# B&R Automation Studio project TD52 (part 136)

#### MSC_MB.st
```iecst
(********************************************************************
 * COPYRIGHT -- INNIO, MSC
 ********************************************************************
 * Library: MSC_MB
 * File: MSC_MB.st
 * Author: Hohensinner Michael
 * Created: April 29, 2021
 ********************************************************************
 * Functions and function blocks of library MSC_MB
 ********************************************************************)
(* ModBus Master function block 4 easy use *)
FUNCTION MSC_MB_RegUpdate
	MSC_MB_RegUpdate := 0;
	bError := FALSE;
	IF tSlave.bSkip THEN
		iWrite	:=	0;
		iRead	:=	0;
		FOR x:=0 TO _MB_CMD_MAX DO
			tSlave.tLine[x].tIF.bExec	:=	FALSE;
		END_FOR
		RETURN;
	END_IF
	FOR x:=0 TO _MB_CMD_MAX DO
		IF tSlave.tLine[x].tDef.pDest > 0 THEN
			CASE tSlave.tLine[x].tDef.iFC OF
				1,2,5,15:	iByteSize := 2 * REAL_TO_UINT(brmceil((UINT_TO_REAL(tSlave.tLine[x].tDef.iLen) + USINT_TO_REAL(tSlave.tLine[x].tDef.iBitOffs))/16.0));		//Bitwise
				3,4,6,16:	iByteSize := 2 * REAL_TO_UINT(brmceil(UINT_TO_REAL(tSlave.tLine[x].tDef.iLen) + USINT_TO_REAL(tSlave.tLine[x].tDef.iBitOffs)/16.0));		//Wordwise
				ELSE
					MSC_MB_RegUpdate := 1;
					RETURN;	// Wrong function code
			END_CASE
			IF SIZEOF(iTemp) < iByteSize THEN
				MSC_MB_RegUpdate := 2;
				RETURN;	// To small temporary register
			END_IF
			IF iByteSize < 2 THEN
				MSC_MB_RegUpdate := 3;
				RETURN;	// To small, at least a word to copy (should not happen)
			END_IF
			brsmemcpy(ADR(iTemp),tSlave.tLine[x].tDef.pDest,iByteSize);

			CASE tSlave.tLine[x].tDef.iFC OF
				1..4:
					IF GET_BIT_UINT_ARRAY(x,ADR(iRead)) THEN
						tSlave.tLine[x].tIF.bExec	:=	bEnaRead;
					END_IF
				5,6,15,16:
					IF GET_BIT_UINT_ARRAY(x,ADR(iWrite)) THEN
						tSlave.tLine[x].tIF.bExec	:=	bEnaWrite;
					END_IF
			END_CASE
			IF tSlave.tLine[x].tIF.iStatus <> 0 AND tSlave.tLine[x].tIF.iStatus <> 65535 THEN
				bError := TRUE;
				iError := tSlave.tLine[x].tIF.iStatus;
			END_IF

			CASE tSlave.tLine[x].tDef.iFC OF
				1,2:
					FOR i:= 0 TO  MAX(0,tSlave.tLine[x].tDef.iLen-1) DO
						IF i > _MB_BIN_MAX THEN
							MSC_MB_RegUpdate := tSlave.tLine[x].tDef.iFC * 10 + 1;
							RETURN;	// OUT OF BINARY BOUNDS
						END_IF
						SET_BIT_UINT_ARRAY(tSlave.tLine[x].tIF.bData[i],i + tSlave.tLine[x].tDef.iBitOffs,ADR(iTemp));
					END_FOR
					brsmemcpy(tSlave.tLine[x].tDef.pDest,ADR(iTemp),iByteSize);
				3,4:
					IF tSlave.tLine[x].tDef.iBitOffs = 0 THEN
						brsmemcpy(tSlave.tLine[x].tDef.pDest,ADR(tSlave.tLine[x].tIF.iData),tSlave.tLine[x].tDef.iLen*2);
					ELSE
						FOR i:= 0 TO MAX(0,tSlave.tLine[x].tDef.iLen*16-1) DO
							IF i/16 > _MB_REG_MAX THEN
								MSC_MB_RegUpdate := tSlave.tLine[x].tDef.iFC * 10 + 1;
								RETURN;	// OUT OF REGISTER BOUNDS
							END_IF
							SET_BIT_UINT_ARRAY(GET_BIT_UINT_ARRAY(i,ADR(tSlave.tLine[x].tIF.iData)),i + tSlave.tLine[x].tDef.iBitOffs,ADR(iTemp));
						END_FOR
						brsmemcpy(tSlave.tLine[x].tDef.pDest,ADR(iTemp),iByteSize);
					END_IF

				5,15:
					IF tSlave.tLine[x].tDef.iFC = 5 THEN
						tSlave.tLine[x].tIF.bData[0] := GET_BIT_UINT_ARRAY(tSlave.tLine[x].tDef.iBitOffs,ADR(iTemp));
					ELSIF tSlave.tLine[x].tDef.iFC = 15 THEN
						FOR i:= 0 TO MAX(0, tSlave.tLine[x].tDef.iLen-1) DO
							IF i > _MB_BIN_MAX THEN
								MSC_MB_RegUpdate := tSlave.tLine[x].tDef.iFC * 10 + 1;
								RETURN;	// OUT OF BINARY BOUNDS
							END_IF
							tSlave.tLine[x].tIF.bData[i]	:=	GET_BIT_UINT_ARRAY(i+tSlave.tLine[x].tDef.iBitOffs,ADR(iTemp));
						END_FOR
					END_IF

				6,16:
					IF tSlave.tLine[x].tDef.iBitOffs = 0 THEN
						FOR i:= 0 TO MAX(0,tSlave.tLine[x].tDef.iLen-1) DO
							IF i > _MB_REG_MAX THEN
								MSC_MB_RegUpdate := tSlave.tLine[x].tDef.iFC * 10;
								RETURN;	// OUT OF REGISTER BOUNDS
							END_IF
							tSlave.tLine[x].tIF.iData[i]	:=	iTemp[i];
						END_FOR
					ELSE
						FOR i:= 0 TO MAX(0,tSlave.tLine[x].tDef.iLen*16-1) DO
							IF i/16 > _MB_REG_MAX THEN
								MSC_MB_RegUpdate := tSlave.tLine[x].tDef.iFC * 10 + 1;
								RETURN;	// OUT OF REGISTER BOUNDS
							END_IF
							SET_BIT_UINT_ARRAY(GET_BIT_UINT_ARRAY(i+tSlave.tLine[x].tDef.iBitOffs,ADR(iTemp)),i,ADR(tSlave.tLine[x].tIF.iData));
						END_FOR
					END_IF
			END_CASE
		END_IF
	END_FOR
	IF NOT bError THEN
		iError	:=	0;
	END_IF
	iWrite	:=	0;
	iRead	:=	0;
	RETURN;
END_FUNCTION

FUNCTION_BLOCK MSC_MBMaster
	IF bEnable THEN
		CASE eState OF
			_MB_DEFAULT:
				IF tCmd.bOpen THEN
					tCmd.bOpen	:=	FALSE;
					eState		:=	_MB_OPEN;
				END_IF
			_MB_OPEN:
				xMBMOpen.enable		:= TRUE;
				xMBMOpen.pDevice	:= ADR(tCfg.sDevice);
				xMBMOpen.pMode		:= ADR(tCfg.sMode);
				xMBMOpen.pConfig	:= ADR(tCfg.sFile);
				xMBMOpen.timeout	:= tCfg.iTimeOut;
				xMBMOpen.ascii		:= BOOL_TO_USINT(tCfg.bASCII);
				xMBMOpen();
				IF (xMBMOpen.status <> ERR_FUB_BUSY) THEN
					IF (xMBMOpen.status = ERR_OK) THEN
						xMBMaster.enable	:=	TRUE;
						xMBMaster.ident		:=	xMBMOpen.ident;
						eState				:=	_MB_RUN;
					ELSE
						eError				:=	eState;
						iError				:=	xMBMOpen.status;
						eState				:=	_MB_ERROR;
					END_IF
				END_IF
			_MB_RUN:
				IF tCmd.bClose THEN
					tCmd.bClose			:=	FALSE;
					xMBMaster.enable	:=	FALSE;
					xMBMClose.enable	:=	TRUE;
					xMBMClose.ident		:=	xMBMOpen.ident;
					eState 				:=	_MB_CLOSE;
				ELSE
					xMBMaster();
				END_IF
			_MB_CLOSE:
				xMBMClose();
				IF (xMBMClose.status <> ERR_FUB_BUSY) THEN
					IF (xMBMClose.status = ERR_OK) THEN
						eState		:=	_MB_DEFAULT;
					ELSE
						eError		:=	eState;
						iError		:=	xMBMOpen.status;
						eState		:=	_MB_ERROR;
					END_IF
				END_IF
			_MB_ERROR:
				IF tCmd.bAckn THEN
					tCmd.bAckn		:=	FALSE;
					eState			:=	_MB_DEFAULT;
				END_IF
		END_CASE
	END_IF
	bExec	:=	xMBMaster.execute;
	iRecNum	:=	xMBMaster.recordnum;
	iStatus	:=	xMBMaster.status;
END_FUNCTION_BLOCK
(* ModBus Slave function block 4 easy use *)
FUNCTION_BLOCK MSC_MBSlave
	IF bEnable THEN
		CASE eState OF
			_MB_DEFAULT:
				IF tCmd.bOpen THEN
					tCmd.bOpen	:=	FALSE;
					eState		:=	_MB_OPEN;
				END_IF
			_MB_OPEN:
				xMBSOpen.enable		:= TRUE;
				xMBSOpen.pDevice	:= ADR(tCfg.sDevice);
				xMBSOpen.pMode		:= ADR(tCfg.sMode);
				xMBSOpen.own_ID		:= tCfg.iID;
				xMBSOpen.timeout	:= tCfg.iTimeOut;
				xMBSOpen.pCoilStat	:= tCfg.pCoilStat;
				xMBSOpen.pHoldingReg:= tCfg.pHoldReg;
				xMBSOpen.pInputReg	:= tCfg.pInReg;
				xMBSOpen.pInputStat	:= tCfg.pInStat;
				xMBSOpen();
				IF (xMBSOpen.status <> ERR_FUB_BUSY) THEN
					IF (xMBSOpen.status = ERR_OK) THEN
						xMBSlave.enable	:=	TRUE;
						xMBSlave.ident		:=	xMBSOpen.ident;
						eState				:=	_MB_RUN;
					ELSE
						eError				:=	eState;
						iError				:=	xMBSOpen.status;
						eState				:=	_MB_ERROR;
					END_IF
				END_IF
			_MB_RUN:
				IF tCmd.bClose THEN
					tCmd.bClose			:=	FALSE;
					xMBSlave.enable		:=	FALSE;
					xMBSClose.enable	:=	TRUE;
					xMBSClose.ident		:=	xMBSOpen.ident;
					eState 				:=	_MB_CLOSE;
				ELSE
					xMBSlave();
				END_IF
			_MB_CLOSE:
				xMBSClose();
				IF (xMBSClose.status <> ERR_FUB_BUSY) THEN
					IF (xMBSClose.status = ERR_OK) THEN
						eState		:=	_MB_DEFAULT;
					ELSE
						eError		:=	eState;
						iError		:=	xMBSOpen.status;
						eState		:=	_MB_ERROR;
					END_IF
				END_IF
			_MB_ERROR:
				IF tCmd.bAckn THEN
					tCmd.bAckn		:=	FALSE;
					eState			:=	_MB_DEFAULT;
				END_IF
		END_CASE
	END_IF
END_FUNCTION_BLOCK

(* ModBus Data Object single line *)
FUNCTION_BLOCK MSC_MB_DataLine
	(* clear old data if previously used *)
	FOR iBegin:=0 TO _MB_DATALINE_MAX DO
		iData[iBegin]	:=	0;
	END_FOR
	bError	:=	FALSE;
	iBegin	:=	0;
	iStrLen	:=	0;
	sData	:=	'';
	(* Execution variable BEGIN *)
	brsstrcat(ADR(sData),ADR('"'));
	IF pName_Module > 0 THEN
		brsstrcat(ADR(sData),pName_Module);
		brsstrcat(ADR(sData),ADR('::'));
	END_IF
	IF pName_Task > 0 THEN
		brsstrcat(ADR(sData),pName_Task);
		brsstrcat(ADR(sData),ADR(':'));
	END_IF
	IF pName_Struct > 0 THEN
		brsstrcat(ADR(sData),pName_Struct);
	ELSE
		brsstrcat(ADR(sData),ADR('tSlave'));
	END_IF
	brsitoa(iIdx_Slave,ADR(sTemp));
	brsstrcat(ADR(sData),ADR('['));
	brsstrcat(ADR(sData),ADR(sTemp));
	brsstrcat(ADR(sData),ADR(']'));

	brsstrcat(ADR(sData),ADR('.tLine'));
	brsitoa(iIdx_Line,ADR(sTemp));
	brsstrcat(ADR(sData),ADR('['));
	brsstrcat(ADR(sData),ADR(sTemp));
	brsstrcat(ADR(sData),ADR('].tIF.bExec"'));

	iStrLen := brsstrlen(ADR(sData))-2;
	IF iStrLen < _MB_DATALINE_MAX THEN
		brsmemcpy(ADR(iData[0]),ADR(sData)+1,iStrLen);
	ELSE
		bError	:=	TRUE;
	END_IF
	(* Execution variable END *)

	(* Spacing *)
	iData[iStrLen] := 0;
	(* Functional code *)
	iData[iStrLen+1] := iFC;
	(* Address of slave *)
	iData[iStrLen+2] := iAdr_Slave;
	iBegin := iStrLen+3;

	(* Data variable BEGIN *)
	sData := '';
	brsstrcat(ADR(sData),ADR('"'));
	IF pName_Module > 0 THEN
		brsstrcat(ADR(sData),pName_Module);
		brsstrcat(ADR(sData),ADR('::'));
	END_IF
	IF pName_Task > 0 THEN
		brsstrcat(ADR(sData),pName_Task);
		brsstrcat(ADR(sData),ADR(':'));
	END_IF
	IF pName_Struct > 0 THEN
		brsstrcat(ADR(sData),pName_Struct);
	ELSE
		brsstrcat(ADR(sData),ADR('tSlave'));
	END_IF

	brsitoa(iIdx_Slave,ADR(sTemp));
	brsstrcat(ADR(sData),ADR('['));
	brsstrcat(ADR(sData),ADR(sTemp));
	brsstrcat(ADR(sData),ADR(']'));

	brsstrcat(ADR(sData),ADR('.tLine'));
	brsitoa(iIdx_Line,ADR(sTemp));
	brsstrcat(ADR(sData),ADR('['));
	brsstrcat(ADR(sData),ADR(sTemp));
	brsstrcat(ADR(sData),ADR('].tIF.'));

	CASE iFC OF
		1,2,15:	brsstrcat(ADR(sData),ADR('bData'));
		3,4,16:	brsstrcat(ADR(sData),ADR('iData'));
		5:	brsstrcat(ADR(sData),ADR('bData[0]'));
		6:	brsstrcat(ADR(sData),ADR('iData[0]'));
		ELSE
			brsstrcat(ADR(sData),ADR('bNA'));	//through error here
	END_CASE
	brsstrcat(ADR(sData),ADR('"'));
	iStrLen := brsstrlen(ADR(sData))-2;
	IF iBegin + iStrLen + 4 < _MB_DATALINE_MAX THEN
		brsmemcpy(ADR(iData[iBegin]),ADR(sData)+1,iStrLen);
		(* Data variable END *)

		(* Spacing *)
		iData[iBegin + iStrLen] := 0;

		(* Offset *)
		iData[iBegin + iStrLen + 1] := UDINT_TO_USINT(iOffset MOD 256);
		iData[iBegin + iStrLen + 2] := UDINT_TO_USINT(iOffset / 256);
		iStrLen	:=	iBegin + iStrLen + 2 + 1;

		(* Length *)
		iData[iStrLen] := UDINT_TO_USINT(iLength MOD 256);
		iData[iStrLen+1] := UDINT_TO_USINT(iLength / 256);
		iStrLen	:=	iStrLen + 2;
	ELSE
		bError	:=	TRUE;
	END_IF

END_FUNCTION_BLOCK

(* ModBus Data Object multiple lines *)
FUNCTION_BLOCK MSC_MB_DataSet
	(* clear old data if previously used *)
	iStrLen	:=	0;
	bError	:=	FALSE;
	FOR i:=0 TO _MB_DATASET_MAX DO
		iData[i]	:=	0;
	END_FOR

	(* handle over static slave data *)
	xLine.pName_Module	:=	pName_Module;
	xLine.pName_Task	:=	pName_Task;
	xLine.pName_Struct	:=	pName_Struct;
	xLine.iIdx_Slave	:=	iIdx_Slave;
	xLine.iAdr_Slave	:=	iAdr_Slave;
	bEmpty	:=	TRUE;

	(* handle over dynamic slave data, execute only if function code is legit *)
	FOR i:= 0 TO _MB_CMD_MAX DO
		IF (tLine[i].tDef.iFC >= 1 AND tLine[i].tDef.iFC <= 6) OR tLine[i].tDef.iFC = 15 OR tLine[i].tDef.iFC = 16	THEN
			xLine.iIdx_Line	:=	UDINT_TO_USINT(i);
			xLine.iFC		:=	tLine[i].tDef.iFC;
			xLine.iOffset	:=	tLine[i].tDef.iOffs;
			xLine.iLength	:=	tLine[i].tDef.iLen;

			xLine();

			IF iStrLen + xLine.iStrLen < _MB_DATASET_MAX AND NOT xLine.bError THEN
				brsmemcpy(ADR(iData)+iStrLen,ADR(xLine.iData),xLine.iStrLen);
				iStrLen	:=	iStrLen + xLine.iStrLen;
				bEmpty	:=	FALSE;
			ELSE
				bError	:=	TRUE;
			END_IF
		END_IF
	END_FOR

END_FUNCTION_BLOCK

(* ModBus Data Object creator *)
FUNCTION_BLOCK MSC_MB_DOCreate

	CASE eState OF
		_MB_DEFAULT:
			xDatObjInfo.enable		:=	TRUE;
			xDatObjInfo.pName 		:=	pName;
			xDatObjDelete.enable	:=	TRUE;
			xDatObjCreate.enable	:=	TRUE;
			xDatObjCreate.pName		:=	pName;
			xDatObjCreate.pCpyData	:=	pCpyData;
			xDatObjCreate.MemType	:=	iMemType;
			xDatObjCreate.len		:=	iLen;
			IF bEnable THEN
				eState	:=	_MB_INFO;
			END_IF
			bDone := FALSE;
		_MB_INFO:
			xDatObjInfo();
			IF	xDatObjInfo.status = ERR_OK THEN				eState	:=	_MB_DELETE;
			ELSIF xDatObjInfo.status = doERR_MODULNOTFOUND THEN	eState	:=	_MB_CREATE;
			ELSIF xDatObjInfo.status <>  ERR_FUB_BUSY THEN		eState	:=	_MB_ERROR;
			END_IF
		_MB_DELETE:
			xDatObjDelete.ident		:=	xDatObjInfo.ident;
			xDatObjDelete();
			IF	xDatObjDelete.status = ERR_OK THEN				eState	:=	_MB_CREATE;
			ELSIF	xDatObjDelete.status <>  ERR_FUB_BUSY THEN	eState	:=	_MB_ERROR;
			END_IF
		_MB_CREATE:
			xDatObjCreate();
			IF	xDatObjCreate.status = ERR_OK THEN				eState	:=	_MB_DONE;
			ELSIF	xDatObjCreate.status <>  ERR_FUB_BUSY THEN	eState	:=	_MB_ERROR;
			END_IF
		_MB_DONE:
			eState;
			bDone := TRUE;
		_MB_ERROR:
			eState;
	END_CASE

END_FUNCTION_BLOCK

(* ModBus Master function block 4 easiest use without data object *)
FUNCTION_BLOCK MSC_MBDOMaster
	CASE eState OF
		_MB_DEFAULT:
			eError	:=	eState;
			IF tCfg.iID > 0 THEN	eState	:=	_MB_START; END_IF
		_MB_START:
			eError	:=	eState;
			xMB_DataSet.pName_Module	:=	pName_Module;
			xMB_DataSet.pName_Task		:=	pName_Task;
			xMB_DataSet.pName_Struct	:=	pName_Struct;

			iLen	:=	0;
			bError	:=	FALSE;
			FOR i:=0 TO _MB_SLAVES_MAX DO
				IF tSlave[i].iMaster = tCfg.iID THEN
					xMB_DataSet.iIdx_Slave	:=	INT_TO_USINT(i);
					xMB_DataSet.iAdr_Slave	:=	tSlave[i].iAdr;
					xMB_DataSet.tLine		:=	tSlave[i].tLine;
					xMB_DataSet();

					IF iLen + xMB_DataSet.iStrLen < _MB_DATAOBJ_MAX AND NOT xMB_DataSet.bError AND xMB_DataSet.iStrLen > 0 AND NOT xMB_DataSet.bEmpty THEN
						brsmemcpy(ADR(iData[iLen]),ADR(xMB_DataSet.iData),xMB_DataSet.iStrLen-1);
						iLen					:=	iLen + xMB_DataSet.iStrLen;
					ELSIF NOT xMB_DataSet.bEmpty THEN
						bError	:=	TRUE;
					END_IF
				END_IF
			END_FOR
			IF NOT bError THEN
				xMB_DOCreate.bEnable		:=	TRUE;
				xMB_DOCreate.pName 			:=	ADR(tCfg.sFile);
				xMB_DOCreate.pCpyData		:=	ADR(iData);
				xMB_DOCreate.iLen			:=	iLen;
				xMB_DOCreate.iMemType		:=	iMemType;
				eState	:=	_MB_CREATE;
			ELSE
				eState	:=	_MB_ERROR;
			END_IF
		_MB_CREATE:
			eError	:=	eState;
			xMB_DOCreate();
			IF xMB_DOCreate.bDone THEN
				eState	:=	_MB_CONFIG;
			END_IF
			IF xMB_DOCreate.eState = _MB_ERROR THEN
				eState	:=	_MB_ERROR;
			END_IF
		_MB_CONFIG:
			eError	:=	eState;
			xMB_Master.bEnable			:=	TRUE;
			xMB_Master.tCfg				:=	tCfg;
			xMB_Master.tCmd				:=	pCmd;
			iEntry						:=	0;
			bError						:=	FALSE;
			FOR i:=0 TO _MB_SLAVES_MAX DO
				IF tSlave[i].iMaster = tCfg.iID THEN
					FOR j:=0 TO _MB_CMD_MAX DO
						IF tSlave[i].tLine[j].tDef.iFC > 0 THEN
							iListSlave[iEntry]	:=	INT_TO_USINT(i);
							iListCmd[iEntry]	:=	INT_TO_USINT(j);
							IF iEntry + 1 <= _MB_ENTRIES_MAX THEN
								iEntry			:=	iEntry + 1;
							ELSE
								bError			:=	TRUE;
							END_IF
						END_IF
					END_FOR
				END_IF
			END_FOR
			IF bError OR iEntry = 0 THEN
				eState	:=	_MB_ERROR;
			ELSE
				eState	:=	_MB_WAIT;
			END_IF
		_MB_WAIT:
			eError	:=	eState;
			IF bEnable THEN	eState	:=	_MB_RUN; END_IF
			FOR i:=0 TO _MB_SLAVES_MAX DO
				iLog[i]	:=	0;
			END_FOR
		_MB_RUN:
			eError	:=	eState;
			FOR i:= 0 TO USINT_TO_INT(iEntry) DO						//skip command accelerator
				iRecNum_Old :=	xMB_Master.iRecNum;
				xMB_Master();
				IF xMB_Master.iRecNum > 0 THEN
					tSlave[iListSlave[xMB_Master.iRecNum-1]].tLine[iListCmd[xMB_Master.iRecNum-1]].tIF.iStatus	:=	xMB_Master.iStatus;
					IF xMB_Master.iStatus > 0 AND xMB_Master.iStatus < ERR_FUB_BUSY THEN
						iLog[iListSlave[xMB_Master.iRecNum-1]]	:=	xMB_Master.iStatus;
					END_IF
					IF iRecNum_Old = xMB_Master.iRecNum THEN EXIT; END_IF
				ELSE
					EXIT;
				END_IF
			END_FOR
			FOR i:=0 TO _MB_SLAVES_MAX DO
				IF xTON_Reset_Log[i].Q THEN
					iLog[i]	:=	0;
				END_IF
				xTON_Reset_Log[i](IN:= iLog[i] <> 0, PT:=T#5s);
			END_FOR
		_MB_ERROR:
			eState;
			eError;
	END_CASE
	bExec	:=	xMB_Master.bExec;
	iRecNum	:=	xMB_Master.iRecNum;
	iStatus	:=	xMB_Master.iStatus;
END_FUNCTION_BLOCK

FUNCTION MSC_MB_DataCheck
	MSC_MB_DataCheck	:=	0;
	FOR i:=0 TO _MB_SLAVES_MAX DO
		//		IF tSlave[i].iMaster > _MB_DEVICES_MAX + 1 THEN
		//			MSC_MB_DataCheck	:=	99;
		//			RETURN;
		//		END_IF
		FOR j:=0 TO _MB_CMD_MAX DO
			CASE tSlave[i].tLine[j].tDef.iFC OF
				1,2,15:
					IF tSlave[i].tLine[j].tDef.iLen > _MB_BIN_MAX + 1 THEN
						MSC_MB_DataCheck	:=	tSlave[i].tLine[j].tDef.iFC;
						RETURN;
					END_IF
				3,4,16:
					IF tSlave[i].tLine[j].tDef.iLen > _MB_REG_MAX + 1 THEN
						MSC_MB_DataCheck	:=	tSlave[i].tLine[j].tDef.iFC;
						RETURN;
					END_IF
				5,6:
					IF tSlave[i].tLine[j].tDef.iLen <> 1 THEN
						MSC_MB_DataCheck	:=	20246;
						RETURN;
					END_IF
				ELSE
					IF tSlave[i].tLine[j].tDef.iFC > 0 THEN
						MSC_MB_DataCheck	:=	tSlave[i].tLine[j].tDef.iFC;
						RETURN;
					END_IF
			END_CASE
		END_FOR
	END_FOR
	RETURN;
END_FUNCTION

FUNCTION UINT_TWO_UDINT
	UINT_TWO_UDINT := UINT_TO_UDINT(IN1)*65536+UINT_TO_UDINT(IN2);
	RETURN;
END_FUNCTION

FUNCTION UINT_TWO_REAL
	brsmemcpy(ADR(UINT_TWO_REAL)+2,ADR(IN1),2);
	brsmemcpy(ADR(UINT_TWO_REAL),ADR(IN2),2);
	RETURN;
END_FUNCTION

FUNCTION STEP
	STEP := DINT_TO_REAL(REAL_TO_DINT(IN/STEPSIZE))*STEPSIZE;
	RETURN;
END_FUNCTION

FUNCTION_BLOCK WAIT_CYCLIC
	IF IN = 0 THEN
		CNT := 0;
		Q := FALSE;
	ELSE
		Q := CNT > IN;
		CNT := CNT+1;
	END_IF
END_FUNCTION_BLOCK

FUNCTION GET_BIT_UINT_ARRAY
	GET_BIT_UINT_ARRAY	:=	(iArray[iBit / 16] AND SHL(1,UINT_TO_SINT(iBit MOD 16))) > 0;
	RETURN;
END_FUNCTION

FUNCTION SET_BIT_UINT_ARRAY
	IF iBit / 16 > _MB_DATA_ARRAY_MAX THEN
		SET_BIT_UINT_ARRAY := TRUE;
		RETURN;
	END_IF
	IF bSet THEN
		iArray[iBit / 16]	:=	iArray[iBit / 16] OR SHL(1,UINT_TO_SINT(iBit MOD 16));
	ELSE
		iArray[iBit / 16]	:=	iArray[iBit / 16] AND NOT SHL(1,UINT_TO_SINT(iBit MOD 16));
	END_IF
	RETURN;
END_FUNCTION
```

#### MSC_MB.typ - Local data types
```iecst
(********************************************************************
 * COPYRIGHT -- INNIO, MSC
 ********************************************************************
 * Library: MSC_MB
 * File: MSC_MB.typ
 * Author: Hohensinner Michael
 * Created: April 29, 2021
 ********************************************************************
 * Functions and function blocks of library MSC_MB
 ********************************************************************)

TYPE
	MB_Reg_Definition : {REDUND_UNREPLICABLE} 	STRUCT
		iFC : {REDUND_UNREPLICABLE} USINT; (*Modbus command function code*)
		iLen : {REDUND_UNREPLICABLE} UINT; (*Modbus command length*)
		iOffs : {REDUND_UNREPLICABLE} UINT; (*Modbus command offset*)
		pDest : {REDUND_UNREPLICABLE} UDINT; (*Destination adress*)
		iBitOffs : {REDUND_UNREPLICABLE} USINT; (*Destination Bit offset*)
		iWordOffs : {REDUND_UNREPLICABLE} USINT; (*Destination word offset to get destination adress*)
	END_STRUCT;
	MB_Reg_Interface : 	STRUCT
		bExec : BOOL; (*Modbus command execution*)
		bData : ARRAY[0.._MB_BIN_MAX]OF BOOL; (*Modbus command binary data*)
		iData : ARRAY[0.._MB_REG_MAX]OF UINT; (*Modbus command 2Byte data*)
		iStatus : UINT; (*Modbus command status*)
	END_STRUCT;
	MB_Reg_Line : 	STRUCT
		tDef : {REDUND_UNREPLICABLE} MB_Reg_Definition; (*Modbus command definition*)
		tIF : MB_Reg_Interface; (*Modbus command execution and data*)
	END_STRUCT;
	MB_Reg_Slaves : 	STRUCT
		bSkip : {REDUND_UNREPLICABLE} BOOL; (*Skips slave is TRUE*)
		sName : {REDUND_UNREPLICABLE} STRING[100]; (*Name of slave*)
		iMaster : {REDUND_UNREPLICABLE} USINT; (*Master identification*)
		iInfo : {REDUND_UNREPLICABLE} USINT; (*Slave information*)
		iAdr : {REDUND_UNREPLICABLE} USINT; (*Station number of slave*)
		tLine : ARRAY[0.._MB_CMD_MAX]OF MB_Reg_Line; (*Modbus command and data*)
	END_STRUCT;
	MBS_Config : {REDUND_UNREPLICABLE} 	STRUCT
		sDevice : {REDUND_UNREPLICABLE} STRING[40]; (*Device adress*)
		sMode : {REDUND_UNREPLICABLE} STRING[40]; (*Modbus mode*)
		iID : {REDUND_UNREPLICABLE} USINT; (*Modbus ID of slave*)
		pInStat : {REDUND_UNREPLICABLE} UDINT; (*Pointer to input status*)
		pInReg : {REDUND_UNREPLICABLE} UDINT; (*Pointer to input register*)
		pHoldReg : {REDUND_UNREPLICABLE} UDINT; (*Pointer to holding register*)
		pCoilStat : {REDUND_UNREPLICABLE} UDINT; (*Pointer to coil status*)
		iTimeOut : {REDUND_UNREPLICABLE} UINT; (*Timeout after X ms*)
	END_STRUCT;
	MBM_Config : {REDUND_UNREPLICABLE} 	STRUCT
		sDevice : {REDUND_UNREPLICABLE} STRING[50]; (*Device adress*)
		sMode : {REDUND_UNREPLICABLE} STRING[40]; (*Modbus mode*)
		sFile : {REDUND_UNREPLICABLE} STRING[40]; (*Dataobject name*)
		bASCII : {REDUND_UNREPLICABLE} BOOL; (*If true ASCII mode is enabled*)
		iTimeOut : {REDUND_UNREPLICABLE} UINT; (*Timeout after X ms*)
		iID : {REDUND_UNREPLICABLE} USINT; (*Master identification number*)
	END_STRUCT;
	MB_Commands : {REDUND_UNREPLICABLE} 	STRUCT
		bOpen : {REDUND_UNREPLICABLE} BOOL; (*Opens modbus communication to the slaves*)
		bClose : {REDUND_UNREPLICABLE} BOOL; (*Closes modbus communication to the slaves*)
		bAckn : {REDUND_UNREPLICABLE} BOOL; (*Acknowledges modbus communication errors*)
	END_STRUCT;
	MB_State_Enum :
		(
		_MB_DEFAULT,
		_MB_OPEN,
		_MB_RUN,
		_MB_CLOSE,
		_MB_START,
		_MB_CREATE,
		_MB_CONFIG,
		_MB_INFO,
		_MB_DELETE,
		_MB_DONE,
		_MB_WAIT,
		_MB_ERROR
		);
	LV_GCB :
		(
		_GCB_INIT,
		_GCB_TRY_ABB,
		_GCB_TRY_SE,
		_GCB_IDLE,
		_GCB_WAIT,
		_GCB_CALC,
		_GCB_CLEAR,
		_ABB_LOAD,
		_ABB_READ,
		_ABB_SAVE_OPEN,
		_ABB_SAVE_DATA,
		_ABB_SAVE_CLOSE,
		_SE_LOAD,
		_SE_READ,
		_SE_SAVE_CHECK,
		_SE_SAVE_CLOSE_OLD,
		_SE_SAVE_OPEN,
		_SE_SAVE_ID,
		_SE_SAVE_DATA1,
		_SE_SAVE_DATA2,
		_SE_SAVE_DATA3,
		_SE_SAVE_APPLY,
		_SE_SAVE_CLOSE,
		_SE_SAVE_CLOSE_CHECK
		);
END_TYPE
```

#### MSC_MB.var
```iecst
VAR CONSTANT
	_MB_DATA_ARRAY_MAX : UINT := 500; (*Maximum size of Data Array*)
	_MB_DEVICES_MAX : USINT := 0; (*Maximum number(+1) of Masters, increase if needed*)
	_MB_SLAVES_MAX : USINT := 1; (*Maximum number(+1) of Slaves, increase if needed*)
	_MB_ENTRIES_MAX : USINT := 159; (*Maximum number(+1) of Commands per Master, increase if needed*)
	_MB_CMD_MAX : USINT := 14; (*Maximum number(+1) of Commands per Slave, increase if needed*)
	_MB_REG_MAX : USINT := 14; (*Maximum number(+1) of Register Data per Command, increase if needed*)
	_MB_BIN_MAX : USINT := 0; (*Maximum number(+1) of Binary Data per Command, increase if needed*)
	_MB_DATALINE_MAX : UDINT := 200; (*Maximum Bytes per data line*)
	_MB_DATASET_MAX : UDINT := 2000; (*Maximum Bytes per slave*)
	_MB_DATAOBJ_MAX : UDINT := 10000; (*Maximum Bytes per master*)
END_VAR
```

### Package Logical/ThermalReactor - TR: Thermo Reactor

### Data object Logical/ThermalReactor/META_TR (Simple) - MODUL META data file

#### META_TR.dat
```
; *******************************************************************************
; AGGR: Module Meta Data (data module)
;
; This code is confidential and proprietary to the INNIO Company.
; It may not be used in any form, or reproduced in any manner, without the express
; written permission of the INNIO Company.
; Copyright, INNIO Company, 2022
;
; Customized modifications: -
; ------------------------
;
; History:
; -------
; V03.99.00.00	06.03.2013	Weitzer		generated for modular software
; V03.99.02.00	29.05.2013	Zengerer	initial dependencies prepared
; V04.00.00.00	30.01.2014	Denk		new version
; V04.03.00.00	25.09.2014	Denk		Start-up changes first Thermoreactor
;				29.06.2015  Denk		Operation hour for Reactor, Gas Injection and el. Heater
; V04.03.01.00	02.11.2015	Zengerer 	MANDATORYMODULE statement
; V04.07.00.00	27.05.2019	Denk		Adjustments regarding new library versions (JEW_LIB1, JEW_LIB2, JEW_LIB3)
; V04.09.00.00	20.02.2020	Denk		Emissions monitoring, messages 9309, 9042, 9043 added
; V04.10.00.00	24.11.2020	lettenb.	2356,2357,2358 added
; V04.11.00.00	28.01.2022	Perktold	included plant controller upgrade
; V04.12.00.00	19.05.2022	Maran		updated electrical heating elements switching logic and trigger signal for hour counter (bugfix)
; V04.13.00.00	27.03.2023	Maran		updated operating temperature definition and maximum temperature difference monitoring for W3503
; 				28.11.2023	Maran		added auxiliary gas injection monitoring inputs
; V04.14.00.00	27.11.2024	Maran		updates for thermal reactor 2nd generation
; 				27.11.2024	Maran		added auxiliary gas stop due to sufficient temperature
; 				27.11.2024	Maran		temperature setpoint reference used in reactor task changed from heating controller out structure value to HMI parameter value
;
; Instructions for use:
; --------------------
; make only changes at the version numbers
;
; Outstandings:
; ------------
;
; *******************************************************************************
;
"<META>"
;
; Module ID
"<MODUL>TR</MODUL>"
;
; Module Version (xx.yy.zz.cc)
"<VERSION>04.14.00.00</VERSION>"
;
; Module Basisupdate Version BU (00-99)
"<BASISUPDATE_VERSION>00</BASISUPDATE_VERSION>"
;
; Optional: specify order number for limitated module usage
"<ORDER></ORDER>" ;<!--(optional for restricted customizations; missing statement makes module valid for all orders)-->
;
; Parameter Check <PARAn Name='aAbcdef' MIN='xxx' MAX='yyy' />  (watch for correct spacings and apostrophs!)
"<PARAMETER_CHK>"
"<PARA1 Name='rT_ThR_EH_Lim75' MIN='1' MAX='800' />"
"<PARA2 />"
"<PARA3 />"
"<PARA4 />"
"<PARA5 />"
"</PARAMETER_CHK>"
;
; Statement, if engine operation is also allowed without this module (FALSE) or if this module´s parameter check passing is mandatory (TRUE)
"<MANDATORYMODULE>FALSE</MANDATORYMODULE>"
;
; Permanent Datamodule Filenames<!-- NAME ist ohne Dateiendung einzutragen; Nur für Counter und interne Parameter verwenden-->
"<DATAMODULES>" ;<!-- optional; mehrere DATAMODULES erlaubt-->
"	<DATAMODULE>par_TR</DATAMODULE>"
"	<DATAMODULE>perm_TR</DATAMODULE>"
"</DATAMODULES>"
;
; Dependencies Modules (MMxx.yy.zz.cc)
"<DEPENDENCIES>"
"	<DEPENDENCY MODULE='AB' VERSION='4.00.00.00' />"
"	<DEPENDENCY MODULE='PB' VERSION='4.00.00.00' />"
"	<DEPENDENCY MODULE='HA' VERSION='4.14.00.00' />"
"	<DEPENDENCY MODULE='OP' VERSION='4.00.00.00' />"
"   <DEPENDENCY VISVERSION='02.15.00.00' />"			; Dependencies Visualization
"</DEPENDENCIES>"
;
; Module function description
"<MODULEFUNCTION>" ;<!-- short overview documentation of module function; add reference to detailed information, if available-->
"	<General>	"
"  Thermal Reactor/CL.AIR module control the operation of the exhaust gas treatment to reduce HCHO and CO emmisions "
"	</General>	"
""
"	<F1 Name='Electric Heater' LastModified='4.14.0.0'>"
"	Electric heater operating power set point "
"	</F1>"
"	<F2 Name='Gas injection' LastModified='4.14.0.0'>"
"	Controls the gas injection valves if available on the Thermal Reactor.	"
"	Monitors the auxiliary gas injection equipment if corresponding instrumentation is available.	"
"	</F2>"
"	<F3 Name='Recirculating valve control' LastModified='4.00.0.0'>"
"	Controls the mixing of the cleaned exhaust gas and the exhaust gas from the cylinder. "
"	</F3>"
"	<F4 Name='Monitoring' LastModified='4.14.0.0'>"
"	 Temperature sensor failure, pressurized air failure, valve end position failure, heat up failure, control panel high temperature, "
"	 high temperature difference within TK1 or TK2, reactor temperature maximum, minimum temperature, operating switch and emission monitoring active "
"	</F4>"
""
"	<Info>"
"	Please enter additional module info here.	"
"	</Info>"
""
"	<Customized LastModified='4.00.0.0'>	"
"	- Nothing "
"	</Customized>	"
""
"</MODULEFUNCTION>"
;
"</META>"
```

### Module_TR.typ - Module global data types
```iecst
TYPE
	IN_TR_Struct : 	STRUCT  (* *) (*OldName: new pv; Cycle:5;*)
		tAB2TR : AmmBase2MM; (*Structure Alarm base to Thermal Reactor module*) (*OldName: new pv; Cycle:5;*)
		tPB2MM : ParaBase2MM_type; (*Data exchange structure to ParaBase*) (*OldName:new PV;Cycle:5*)
		tEng_Run : HALioDo_Type; (*Engine in operation*) (*OldName:M_BTRB;Cycle:5*)
		iSt_OpMode : UDINT; (*Operating mode*) (*OldName:new pv; Cycle:5;*)
		tThR_LampTest : HALioDi_Type; (* DI thermal reactor lamp test *) (*OldName:DI_LT; Cycle:5;*)
		tThR_SL : HALioDi_Type; (* DI thermal reactor safety loop *) (*OldName:DI_SIK_TH; Cycle:5;*)
		tThR_Swth_On : HALioDi_Type; (* DI thermal reactor operation switch on *) (*OldName:DI_S_EIN; Cycle:5;*)
		tGCB_On : HALioDi_Type; (* generator circuit breaker closed *) (*OldName:GCB_ON;Cycle:2*)
		tMCB_On : HALioDi_Type; (* mains circuit breaker closed *) (*OldName:MCB_ON;Cycle:5*)
		tPos_ThR_Val_In1 : HALioDi_Type; (* DI1 thermal reactor flap in position moved in *) (*OldName:DI_KL_EIN1; Cycle:5;*)
		tPos_ThR_Val_In2 : HALioDi_Type; (* DI2 thermal reactor flap in position moved in *) (*OldName:DI_KL_EIN2; Cycle:5;*)
		tPos_ThR_Val_Mid : HALioDi_Type; (* DI thermal reactor flap in middle position *) (*OldName:DI_E_MITT; Cycle:5;*)
		tPos_ThR_Val_Out1 : HALioDi_Type; (* DI1 thermal reactor flap in position moved out *) (*OldName:DI_KL_AUS1; Cycle:5;*)
		tPos_ThR_Val_Out2 : HALioDi_Type; (* DI2 thermal reactor flap in position moved out *) (*OldName:DI_KL_AUS2; Cycle:5;*)
		tPr_ThR_AirLo : HALioDi_Type; (* DI thermal reactor compressed air pressure low *) (*OldName:DI_PS_LUFT; Cycle:5;*)
		tT_ThR_ChamberLo : HALioDi_Type; (* DI thermal reactor chamber temperature low *) (*OldName:DI_T_MIN; Cycle:5;*)
		tT_ThR_Swg_Hi : HALioDi_Type; (* DI thermal reactor switchgear temperature high *) (*OldName:DI_SR_TEMP; Cycle:5;*)
		rP_Act_Norm_Filt : REAL; (* actual power related to rP_Nom filtered T=1s *) (*OldName:P_IST_PROM; Cycle:5;*)
		rP_Nom : REAL; (*Nominal power*) (*OldName:PN_GASART;Cycle:5;*)
		tT_ThR_Chamber1_1 : HALioAi_Type; (* thermal reactor chamber temperature 1_1 *) (*OldName:TK1_1; Cycle:5;*)
		tT_ThR_Chamber1_2 : HALioAi_Type; (* thermal reactor chamber temperature 1_2 *) (*OldName:TK1_2; Cycle:5;*)
		tT_ThR_Chamber2_1 : HALioAi_Type; (* thermal reactor chamber temperature 2_1 *) (*OldName:TK2_1; Cycle:5;*)
		tT_ThR_Chamber2_2 : HALioAi_Type; (* thermal reactor chamber temperature 2_2 *) (*OldName:TK2_2; Cycle:5;*)
		tT_ThR_Comp : HALioAi_Type; (* thermal reactor compensation temperature *) (*OldName:AI_Tvgl; Cycle:5;*)
		tT_ThR_In : HALioAi_Type; (* thermal reactor inlet temperature *) (*OldName:AI_TempInTR; Cycle:5;*)
		tT_ThR_Out : HALioAi_Type; (* thermal reactor outlet temperature *) (*OldName:AI_TempOutTR; Cycle:5;*)
		tTR_AuxPS_GndFault : HALioDi_Type; (*earth fault auxiliaries power supply thermal reactor panel*)
		tTR_AuxPS_CB_Trip : HALioDi_Type; (*auxiliaries power supply circuit breaker thermal reactor panel tripped*)
		tTR_AuxPS_CB_On : HALioDi_Type; (*auxiliaries power supply circuit breaker thermal reactor panel opened*)
		tPos_ThR_AuxGasCV_Act : HALioAi_Type; (* Thermal reactor - auxiliary gas injection control valve position [%] (P.16-S-001) *)
		tPr_ThR_AuxGasBeforeCV : HALioAi_Type; (* Thermal reactor - auxiliary gas pressure before control valve [mbar] (P.16-PI-010) *)
		tPr_ThR_AuxGasAfterCV : HALioAi_Type; (* Thermal reactor - auxiliary gas pressure after control valve [mbar] (P.16-PI-020) *)
		tPr_ThR2_Inlet : HALioAi_Type; (* Thermal reactor 2 - inlet pressure [mbar] (P.02-PI-201) *)
		tPr_ThR2_Outlet : HALioAi_Type; (* Thermal reactor 2 - outlet pressure [mbar] (P.02-PI-202) *)
		tT_ThR2_EH_group1 : HALioAi_Type; (* Thermal reactor 2 - electrical heating group 1 - temperature [degC] (P.16-TI-101) *) (*Cycle:5;*)
		tT_ThR2_EH_group2 : HALioAi_Type; (* Thermal reactor 2 - electrical heating group 2 - temperature [degC] (P.16-TI-201) *) (*Cycle:5;*)
		tT_ThR2_EH_group3 : HALioAi_Type; (* Thermal reactor 2 - electrical heating group 3 - temperature [degC] (P.16-TI-301) *) (*Cycle:5;*)
		tT_ThR2_EH_group4 : HALioAi_Type; (* Thermal reactor 2 - electrical heating group 4 - temperature [degC] (P.16-TI-401) *) (*Cycle:5;*)
		tT_ThR2_EH_group5 : HALioAi_Type; (* Thermal reactor 2 - electrical heating group 5 - temperature [degC] (P.16-TI-501) *) (*Cycle:5;*)
		tT_ThR2_LeftChamber : HALioAi_Type; (* Thermal reactor 2 - chamber temperature left side [degC] (P.16-TI-018) *) (*Cycle:5;*)
		tT_ThR2_RightChamber : HALioAi_Type; (* Thermal reactor 2 - chamber temperature right side [degC] (P.16-TI-017) *) (*Cycle:5;*)
		tT_ThR2_Downstream : HALioAi_Type; (* Thermal reactor 2 - downstream temperature [degC] (P.16-TI-021) *) (*Cycle:5;*)
		tThR2_T_UnitOk_LeftCh : HALioDi_Type; (* Thermal reactor 2 - Sensor processing unit ok - chamber temperature left side (P.16-TI-018) *)
		tThR2_T_UnitOk_RightCh : HALioDi_Type; (* Thermal reactor 2 - Sensor processing unit ok - chamber temperature right side (P.16-TI-017) *)
		tThR2_T_UnitOk_Downstream : HALioDi_Type; (* Thermal reactor 2 - Sensor processing unit ok - downstream temperature (P.16-TI-021) *)
		tPr_SCR_CatIn : HALioAi_Type; (*SCR Exhaust pressure CAT inlet [bar] (P.02-PI-101)*)
	END_STRUCT;
	OUT_TR_Struct : 	STRUCT
		tTR2PB : MM2ParaBase_type; (*Data exchange structure to ParaBase*) (*OldName: new pv; Cycle:5;*)
		tTR2AB : MM2AmmBase; (*AMM Structure*) (*OldName: new pv; Cycle:5;*)
		tThR_Contactor : HALioDo_Type; (* DO thermal reactor contactor *) (*OldName:DO_SCHUETZ; Cycle:5;*)
		tThR_CV_CDec : HALioDo_Type; (* DO thermal reactor gas control valve command decrease *) (*OldName:DO_GAS_MINUS; Cycle:5;*)
		tThR_CV_CInc : HALioDo_Type; (* DO thermal reactor gas control valve command increase *) (*OldName:DO_GAS_PLUS; Cycle:5;*)
		tThR_EH11 : HALioDo_Type; (* DO thermal reactor electrical heating element group 1 output 1 *) (*OldName:b_ThR_EH11; Cycle:5;*)
		tThR_EH12 : HALioDo_Type; (* DO thermal reactor electrical heating element group 1 output 2 *) (*OldName:b_ThR_EH12; Cycle:5;*)
		tThR_EH13 : HALioDo_Type; (* DO thermal reactor electrical heating element group 1 output 3 *) (*OldName:b_ThR_EH13; Cycle:5;*)
		tThR_EH21 : HALioDo_Type; (* DO thermal reactor electrical heating element group 2 output 1 *) (*OldName:b_ThR_EH21; Cycle:5;*)
		tThR_EH22 : HALioDo_Type; (* DO thermal reactor electrical heating element group 2 output 2 *) (*OldName:b_ThR_EH22; Cycle:5;*)
		tThR_EH23 : HALioDo_Type; (* DO thermal reactor electrical heating element group 2 output 3 *) (*OldName:b_ThR_EH23; Cycle:5;*)
		tThR_EH31 : HALioDo_Type; (* DO thermal reactor electrical heating element group 3 output 1 *) (*OldName:b_ThR_EH31; Cycle:5;*)
		tThR_EH32 : HALioDo_Type; (* DO thermal reactor electrical heating element group 3 output 2 *) (*OldName:b_ThR_EH32; Cycle:5;*)
		tThR_EH33 : HALioDo_Type; (* DO thermal reactor electrical heating element group 3 output 3 *) (*OldName:b_ThR_EH33; Cycle:5;*)
		tThR_ErrLamp : HALioDo_Type; (* DO thermal reactor failure lamp *) (*OldName:DO_L_ST; Cycle:5;*)
		tThR_GT_COn1 : HALioDo_Type; (* DO1 thermal reactor gas injection command on *) (*OldName:DO_EIND_EIN1; Cycle:5;*)
		tThR_GT_COn2 : HALioDo_Type; (* DO2 thermal reactor gas injection command on *) (*OldName:DO_EIND_EIN2; Cycle:5;*)
		bThR_RelGas : BOOL; (* thermal reactor gas injection released *) (*OldName:FRG_GASREG; Cycle:5;*)
		bThR_RelGas_Tmin : BOOL; (* thermal reactor minimum temperature for gas injection reached *) (*Cycle:5;*)
		bThR_RelHeat : BOOL; (* thermal reactor heating released *) (*OldName:FG_HEIZG; Cycle:5;*)
		bThR_Run : BOOL; (* thermal reactor operating *) (*OldName:TR_ON; Cycle:5;*)
		tThR_RunLamp : HALioDo_Type; (* DO thermal reactor operating lamp *) (*OldName:DO_L_BETR; Cycle: 5;*)
		bThR_RunReacTemp : BOOL; (* thermal reactor operating on reaction temperature *) (*OldName:TR_OPER; Cycle:5;*)
		tCtrTR_Heater_Set : HALioAo_Type; (*AO -> Controller output*)
		tThR_Val_Air : HALioDo_Type; (* DO thermal reactor purge air valve *) (*OldName:DO_SPLU_STOP; Cycle:5;*)
		tThR_Val_CCylIn : HALioDo_Type; (* DO thermal reactor flap command move in cylinder *) (*OldName:DO_KL_EIN; Cycle:5;*)
		tThR_Val_CCylOut : HALioDo_Type; (* DO thermal reactor flap command move out cylinder *) (*OldName:DO_KL_AUS; Cycle:5;*)
		bThR_Val_SetIn : BOOL; (* thermal reactor flap set direction move in cylinder *) (*OldName:KL_EIN; Cycle:5;*)
		bThR_Val_SetOut : BOOL; (* thermal reactor flap set direction move out cylinder *) (*OldName:KL_AUS; Cycle:5;*)
		bThR_Active : BOOL; (* thermal reactor measuring active *) (*OldName:reactor_a; Cycle:5;*)
		rP_ThR_EH : REAL; (* thermal reactor electrical heating power *) (*OldName:y_HE_Prom; Cycle:5;*)
		rT_ThR_Chamber : REAL; (* thermal reactor chamber temperature *) (*OldName:TK; Cycle:5;*)
		rT_ThR_Chamber1_1 : REAL; (* thermal reactor chamber temperature 1_1 *) (*OldName:TK1_1; Cycle:5;*)
		rT_ThR_Chamber1_2 : REAL; (* thermal reactor chamber temperature 1_2 *) (*OldName:TK1_2; Cycle:5;*)
		rT_ThR_Chamber2_1 : REAL; (* thermal reactor chamber temperature 2_1 *) (*OldName:TK2_1; Cycle:5;*)
		rT_ThR_Chamber2_2 : REAL; (* thermal reactor chamber temperature 2_2 *) (*OldName:TK2_2; Cycle:5;*)
		rT_ThR_Comp : REAL; (* thermal reactor compensation temperature *) (*OldName:Tvgl; Cycle:5;*)
		rT_ThR_In : REAL; (* thermal reactor inlet temperature *) (*OldName:TempInTR; Cycle:5;*)
		rT_ThR_Out : REAL; (* thermal reactor outlet temperature *) (*OldName:TempOutTR; Cycle:5;*)
		tCtrTR_Heater_Out : _tGeACtrOut; (* Heater Controller *) (*OldName: newPV; Cycle:5;*)
		tThR2_EH_group1_Dem : HALioDo_Type; (* Thermal reactor 2 - electrical heating group 1 - command On (P.16-W-101,102,103,104,105) *) (*Cycle:5;*)
		tThR2_EH_group2_Dem : HALioDo_Type; (* Thermal reactor 2 - electrical heating group 2 - command On (P.16-W-201,202,203) *) (*Cycle:5;*)
		tThR2_EH_group3_Dem : HALioDo_Type; (* Thermal reactor 2 - electrical heating group 3 - command On (P.16-W-301,302,303,304,305) *) (*Cycle:5;*)
		tThR2_EH_group4_Dem : HALioDo_Type; (* Thermal reactor 2 - electrical heating group 4 - command On (P.16-W-401,402,403) *) (*Cycle:5;*)
		tThR2_EH_group5_Dem : HALioDo_Type; (* Thermal reactor 2 - electrical heating group 5 - command On (P.16-W-501,502,503,504,505) *) (*Cycle:5;*)
		tThR2_AuxGasShutOffValve_Dem : HALioDo_Type; (* Thermal reactor 2 - solenoid valve gas injection - command Open (P.16-YCS-009) *) (*Cycle:5;*)
	END_STRUCT;
	MM2VIS_Struct : 	STRUCT
		tCtrTR_Heater_Out : _tGeACtrOut; (*Controller to visualization OUT- structure*) (*OldName: newPV; Cycle:5;*)
		b_ThR_Val_Air : BOOL; (*Thermal reactor purge air valve*) (*OldName:DO_SPLU_STOP; Cycle:5;*)
		rP_ThR_EH : REAL; (*Electrical heating power*) (*OldName:y_HE_Prom1; Cycle:5;*)
		bThR_GT_COn2 : BOOL; (*Thermal reactor gas injection valve 2*) (*OldName:DO_EIND_EIN2; Cycle:5;*)
		bThR_GT_COn1 : BOOL; (*Thermal reactor gas injection valve 1*) (*OldName:DO_EIND_EIN1; Cycle:5;*)
		bPos_ThR_Val_Out2 : BOOL; (*Thermal reactor flap in position moved out 2*) (*OldName: DI_KL_AUS2; Cycle: 5;*)
		bPos_ThR_Val_In2 : BOOL; (*Thermal reactor flap in position moved in 2*) (*OldName: DI_KL_EIN2; Cycle: 5;*)
		bPos_ThR_Val_Mid : BOOL; (*Thermal reactor flap in position middle*) (*OldName: DI_KL_MITT; Cycle:5;*)
		bPos_ThR_Val_Out1 : BOOL; (*Thermal reactor flap in position moved out 1*) (*OldName: DI_KL_AUS1; Cycle: 5;*)
		bPos_ThR_Val_In1 : BOOL; (*Thermal reactor flap in position moved in 1*) (*OldName: DI_KL_EIN1; Cycle: 5;*)
		rT_ThR_Out : REAL; (*Thermal reactor outlet temperature*) (*OldName:AI_TempOut; Cycle: 5;*)
		rT_ThR_In : REAL; (*Thermal reactor inlet temperature*) (*OldName:AI_TempIn; Cycle: 5;*)
		rT_ThR_Comp : REAL; (*Thermal reactor compensation temperature*) (*OldName:Tvgl; Cycle:5;*)
		rT_ThR_Chamber : REAL; (*Thermal reactor average chamber temperature*) (*OldName:TK; Cycle:5;*)
		rT_ThR_Chamber2_2 : REAL; (*Thermal reactor chamber temperature 2_2*) (*OldName:TK2_2; Cycle:5;*)
		rT_ThR_Chamber2_1 : REAL; (*Thermal reactor chamber temperature 2_1*) (*OldName:TK2_1; Cycle:5;*)
		rT_ThR_Chamber1_2 : REAL; (*Thermal reactor chamber temperature 1_2*) (*OldName:TK1_2; Cycle:5;*)
		rT_ThR_Chamber1_1 : REAL; (*Thermal reactor chamber temperature 1_2*) (*OldName:TK1_1; Cycle:5;*)
		bMsg3306 : BOOL; (* Disturbance exhasut valvue middle position *) (*OldName:ALM[3306]; Cycle:5;*)
		bMsg3307 : BOOL; (* Safety loop thermal reactor, active only with RIO *) (*OldName:ALM[3307]; Cycle:5;*)
		bMsg3498 : BOOL; (* Sensor failure  *) (*OldName:ALM[3498]; Cycle:5;*)
		bMsg3499 : BOOL; (* Disturbance in pressurized air supply *) (*OldName:ALM[3499]; Cycle:5;*)
		bMsg3500 : BOOL; (* Disturbance in exhasut valve end position *) (*OldName:ALM[3500]; Cycle:5;*)
		bMsg3501 : BOOL; (* Heating time exceeded *) (*OldName:ALM[3501]; Cycle:5;*)
		bMsg3502 : BOOL; (* Control panel temperature too high *) (*OldName:ALM[3502]; Cycle:5;*)
		bMsg3503 : BOOL; (* Temperature differnce between TK1/TK2  > allowed maximum*) (*OldName:ALM[3503]; Cycle:5;*)
		bMsg3504 : BOOL; (* Reactor temperature TK1/TK2 maximum *) (*OldName:ALM[3504]; Cycle:5;*)
		bMsg3505 : BOOL; (* Reactor temperature minimum *) (*OldName:ALM[3505]; Cycle:5;*)
		bThR_RelHeat : BOOL; (* thermal reactor heating released *) (*OldName:FG_HEIZG; Cycle:5;*)
		bThR_Val_SetIn : BOOL; (* thermal reactor flap set direction move in cylinder *) (*OldName:KL_EIN; Cycle:5;*)
		bThR_Val_SetOut : BOOL; (* thermal reactor flap set direction move out cylinder *) (*OldName:KL_AUS; Cycle:5;*)
		bThR_RelGas : BOOL; (* thermal reactor gas injection released *) (*OldName:FRG_GASREG; Cycle:5;*)
		bMsg9309 : BOOL;
		bMsg9042 : BOOL;
		bMsg9043 : BOOL;
		bMsg2356 : BOOL;
		bMsg2357 : BOOL;
		bMsg2358 : BOOL;
		rPos_ThR_AuxGasCV_Act : REAL; (* Thermal reactor - auxiliary gas injection control valve position [%] (P.16-S-001) *)
		rPr_ThR_AuxGasBeforeCV : REAL; (* Thermal reactor - auxiliary gas pressure before control valve [mbar] (P.16-PI-010) *)
		rPr_ThR_AuxGasAfterCV : REAL; (* Thermal reactor - auxiliary gas pressure after control valve [mbar] (P.16-PI-020) *)
		rPr_Diff_ThR_AuxGasCV : REAL; (* Thermal reactor - auxiliary gas differential pressure across control valve [mbar] *)
		bThr_AuxGasCompressor_Run : BOOL; (* Thermal reactor - auxiliary gas compressor derived running status *)
		rFlow_ThR_AuxGasCV : REAL; (* Thermal reactor - calculated auxiliary gas flow (control valve) [Nm3/h] *)
		bMsg9374 : BOOL; (* Measuring signal failure auxiliary gas control valve position *)
		bMsg9375 : BOOL; (* Measuring signal failure auxiliary gas pressure before control valve *)
		bMsg9376 : BOOL; (* Measuring signal failure auxiliary gas pressure after control valve *)
		bMsg9377 : BOOL; (* Thermal reactor - auxiliary gas compressor fault, low pressure before control valve *)
		bMsg9381 : BOOL; (* Thermal reactor - implausible auxiliary gas pressure before/after control valve *)
		bMsg9396 : BOOL; (* Thermal reactor - differential pressure maximum - ThR2 *)
		bMsg9397 : BOOL; (* Measuring signal failure thermal reactor inlet pressure - ThR2 *)
		bMsg9398 : BOOL; (* Measuring signal failure thermal reactor outlet pressure - ThR2 *)
		bMsg9500 : BOOL; (* Measuring signal failure electrical heating monitoring temperature sensors - ThR2 *)
		bMsg9501 : BOOL; (* Measuring signal failure thermal reactor temperature right side - ThR2 *)
		bMsg9502 : BOOL; (* Measuring signal failure thermal reactor temperature left side - ThR2 *)
		bMsg9503 : BOOL; (* Measuring signal failure thermal reactor downstream temperature - ThR2 *)
		bMsg9504 : BOOL; (* Thermal reactor - auxiliary gas injection solenoid valve fault - ThR2 *)
		bMsg9505 : BOOL; (* Exhaust aftertreatment: Thermal reactor outlet/SCR inlet high differential pressure - ThR2 *)
		rPr_ThR2_Inlet : REAL; (* Thermal reactor 2 - inlet pressure [mbar] (P.02-PI-201) *)
		rPr_ThR2_Outlet : REAL; (* Thermal reactor 2 - outlet pressure [mbar] (P.02-PI-202) *)
		rPr_Diff_ThR2 : REAL; (* Thermal reactor 2 - inlet/outlet differential pressure [mbar] *)
		rT_ThR2_LeftChamber : REAL; (* Thermal reactor 2 - chamber temperature left side [degC] (P.16-TI-018) *)
		rT_ThR2_RightChamber : REAL; (* Thermal reactor 2 - chamber temperature right side [degC] (P.16-TI-017) *)
		rT_ThR2_Downstream : REAL; (* Thermal reactor 2 - downstream temperature [degC] (P.16-TI-021) *)
		bThR2_T_fault_LeftCh : BOOL; (* Thermal reactor 2 - Sensor fault - chamber temperature left side (P.16-TI-018) *)
		bThR2_T_fault_RightCh : BOOL; (* Thermal reactor 2 - Sensor fault - chamber temperature right side (P.16-TI-017) *)
		bThR2_T_fault_Downstream : BOOL; (* Thermal reactor 2 - Sensor fault - downstream temperature (P.16-TI-021) *)
		iThR2_EH_group1_status : UINT; (* Thermal reactor 2 - electrical heating group 1 - status (P.16-W-101,102,103,104,105) *)
		iThR2_EH_group2_status : UINT; (* Thermal reactor 2 - electrical heating group 2 - status (P.16-W-201,202,203) *)
		iThR2_EH_group3_status : UINT; (* Thermal reactor 2 - electrical heating group 3 - status (P.16-W-301,302,303,304,305) *)
		iThR2_EH_group4_status : UINT; (* Thermal reactor 2 - electrical heating group 4 - status (P.16-W-401,402,403) *)
		iThR2_EH_group5_status : UINT; (* Thermal reactor 2 - electrical heating group 5 - status (P.16-W-501,502,503,504,505) *)
		rT_ThR2_EH_group1 : REAL; (* Thermal reactor 2 - electrical heating group 1 - temperature [degC]*)
		rT_ThR2_EH_group2 : REAL; (* Thermal reactor 2 - electrical heating group 1 - temperature [degC]*)
		rT_ThR2_EH_group3 : REAL; (* Thermal reactor 2 - electrical heating group 1 - temperature [degC]*)
		rT_ThR2_EH_group4 : REAL; (* Thermal reactor 2 - electrical heating group 1 - temperature [degC]*)
		rT_ThR2_EH_group5 : REAL; (* Thermal reactor 2 - electrical heating group 1 - temperature [degC]*)
		bThR2_AuxGasShutOffValve_Dem : BOOL; (* Thermal reactor 2 - solenoid valve gas injection - command Open (P.16-YCS-009) *)
		bThR_LeftChamber_inlet : BOOL; (* Thermal reactor 2 - left side inlet status *)
		bThR_RightChamber_inlet : BOOL; (* Thermal reactor 2 - right side inlet status  *)
		rPr_Diff_ThR2out_SCRin : REAL; (* Thermal reactor 2 - Exhaust aftertreatment - Thermal reactor outlet/SCR inlet differential pressure [mbar] *)
	END_STRUCT;
	VIS2MM_Struct : 	STRUCT
		tCtrTR_Heater_In : _tGeACtrIn; (*Visualization to controller IN - structure*)
		iCnt_OpHours_Reactor : DINT;
		iCnt_OpHours_GasInj : DINT;
		iCnt_OpHours_Heater : DINT;
	END_STRUCT;
	PERM_TR_Struct : 	STRUCT
		iCnt_OpHours_Reactor : DINT;
		iCnt_OpHours_GasInj : DINT;
		iCnt_OpHours_Heater : DINT;
		rTB_PermValue04 : REAL; (*spare permanent value for testbench- replace with new vars of same lenght, when needed*) (*OldName:new PV;Cycle:2;*)
		rTB_PermValue05 : REAL; (*spare permanent value for testbench- replace with new vars of same lenght, when needed*) (*OldName:new PV;Cycle:2;*)
		rTB_PermValue06 : REAL; (*spare permanent value for testbench- replace with new vars of same lenght, when needed*) (*OldName:new PV;Cycle:2;*)
		rTB_PermValue07 : REAL; (*spare permanent value for testbench- replace with new vars of same lenght, when needed*) (*OldName:new PV;Cycle:2;*)
		rTB_PermValue08 : REAL; (*spare permanent value for testbench- replace with new vars of same lenght, when needed*) (*OldName:new PV;Cycle:2;*)
		rTB_PermValue09 : REAL; (*spare permanent value for testbench- replace with new vars of same lenght, when needed*) (*OldName:new PV;Cycle:2;*)
		rTB_PermValue10 : REAL; (*spare permanent value for testbench- replace with new vars of same lenght, when needed*) (*OldName:new PV;Cycle:2;*)
	END_STRUCT;
	ls : 	STRUCT
		IN : DINT;
		LSHI : DINT;
		LSLO : DINT;
		QH : BOOL;
		QL : BOOL;
	END_STRUCT;
	ls_t : 	STRUCT
		IN : DINT;
		LSHI : DINT;
		LSLO : DINT;
		PTHI : TIME;
		PTLO : TIME;
		QH : BOOL;
		QL : BOOL;
	END_STRUCT;
END_TYPE
```

### Module_TRPara.typ - Module global Parameter data types
```iecst
TYPE
	PROGRAMMER_INFO : 	STRUCT
		DO_NOT_SORT_PARA : STRING[40] := 'DO NOT CHANGE PARAMETER SORTING!'; (*DO NOT CHANGE PARAMETER SORTING!*) (*ADD NEW PARAMETER ONLY AT THE END OF THE Para STRUCTURE. DO NOT DELETE existing Para items.*)
	END_STRUCT;
	Para_Struct : 	STRUCT
		bSel_FlapActEl : BOOL; (*PARA [12749]: select Flap with electric actuation*) (*OldName: sel_FlapActEl;Cycle:5;*)
		bCtrThR_Heater_Active : BOOL; (*PARA [12222]: thermal reactor controller active*) (*OldName: newpv ; Cycle: ;*)
		tCtrTR_Heater : _tGeACtrPara; (*Para controller parameters*) (*OldName: newpv; Cycle: ;*)
		rT_ThR_SetwoGas : REAL; (*PARA [12236]: TK setpoint without gas injection*) (*OldName:TK_w_woGas; Cycle:5;*)
		ti_ThR_Val_y2 : TIME; (*PARA [12241]: timer 2 for exhaust gas flap at TK_w + temperature 2 [s]*) (*OldName:i_ThR_Val_y2; Cycle: 5;*)
		ti_ThR_Val_y1 : TIME; (*PARA [12240]: timer 1 for exhaust gas flap at TK_w + temperature 1 [s]*) (*OldName:i_ThR_Val_y1; Cycle: 5;*)
		ti_ThR_TimePInc : TIME; (*PARA [12239]: time slot load monitoring P increase [s]*) (*OldName:TimeSlot_Pinc; Cycle:5;*)
		bThR_Active : BOOL; (*PARA [12223]: thermal reactor active*) (*OldName:bExhReactor; Cycle:5;*)
		rT_ThR_Val_x2 : REAL; (*PARA [12238]: temperature 2 relative to TK_w for timer 2*) (*OldName:PT_KLrx2; Cycle: 5;*)
		rT_ThR_Val_x1 : REAL; (*PARA [12237]: temperature 1 relative to TK_w for timer 1*) (*OldName:PT_KLrx1; Cycle: 5;*)
		bThR_woGas : BOOL; (*PARA [12225]: select w/o gas injection*) (*OldName:sel_woGas; Cycle: 5;*)
		rP_ThR_ActiveHy : REAL; (*PARA [12227]: power limit thermal reactor active hysteresis*) (*OldName:HY_P_TRACT; Cycle:5;*)
		rP_Norm_ThR_Active : REAL; (*PARA [12226]: power limit norm thermal reactor active (0-100%)*) (*OldName:GW_P_TRACT; Cycle:5;*)
		rT_ThR_LimPInc : REAL; (*PARA [12235]: limit P increase*) (*OldName:Limit_Pinc; Cycle:5;*)
		rT_ThR_LimGasHy : REAL; (*PARA [12234]: limit of reaction chamber temperature for start gas injection hysteresis*) (*OldName:TK_GAS_Hy; Cycle:5;*)
		rT_ThR_LimGas : REAL; (*PARA [12233]: limit of reaction chamber temperature for start gas injection*) (*OldName:TK_GAS_Gw; Cycle:5;*)
		rT_ThR_EH_Lim25 : REAL; (*PARA [12230]: limit of reaction chamber temperature for limitation el. heating to 25% *) (*OldName:TK_E25_Gw; Cycle:5;*)
		rT_ThR_EH_Lim50 : REAL; (*PARA [12231]: limit of reaction chamber temperature for limitation el. heating to 50% *) (*OldName:TK_E50_Gw; Cycle:5;*)
		rT_ThR_EH_Lim75 : REAL; (*PARA [12232]: limit of reaction chamber temperature for limitation el. heating to 75% *) (*OldName:TK_E75_Gw; Cycle:5;*)
		rT_ThR_EH_Lim00 : REAL; (*PARA [12229]: limit of reaction chamber temperature for limitation el. heating to 0% *) (*OldName:TK_E00_Gw; Cycle:5;*)
		ti_ThR_ValDurationPInc : TIME; (*PARA [12242]: duration flap interval increase [s]*) (*OldName:PTOF_KL_Pinc_i; Cycle:5;*)
		ti_ThR_ValIntervalPInc : TIME; (*PARA [12243]: flap interval time increase [s]*) (*OldName:PT_KL_Pinc; Cycle:5;*)
		iIdx_Em_AvgMon_Option : INT; (*PARA [14279]: Emission average monitoring options*)
		bThR_auxGasMonitor : BOOL; (*PARA [14948]: Thermal reactor auxiliary gas injection monitoring *)
		rThR_auxGasCV_Kv : REAL; (*PARA [14949]: Auxiliary gas injection control valve flow coefficient [m3/h]  *)
		bThR2_Ena : BOOL; (*PARA [15036]: Thermal reactor 2nd generation enable *)
		rT_ThR2_EH_Lim00 : REAL; (*PARA [15043]: Thermal reactor chamber temperature for limiting el. Heating to 0% *)
		rT_ThR2_EH_Lim20 : REAL; (*PARA [15040]: Thermal reactor chamber temperature for limiting el. Heating to 20% *)
		rT_ThR2_EH_Lim40 : REAL; (*PARA [15039]: Thermal reactor chamber temperature for limiting el. Heating to 40% *)
		rT_ThR2_EH_Lim60 : REAL; (*PARA [15038]: Thermal reactor chamber temperature for limiting el. Heating to 60% *)
		rT_ThR2_EH_Lim80 : REAL; (*PARA [15037]: Thermal reactor chamber temperature for limiting el. Heating to 80% *)
		bPr_SCR_CatIn_Exist : BOOL; (*PARA [13905]: SCR Exhaust pressure CAT inlet active*)
		bSCR_Active : BOOL; (*PARA [13961]: SCR active*)
		bSCR_Cust_Active : BOOL; (*PARA [14866]: Customer SCR active*)
	END_STRUCT;
END_TYPE
```

### Module_TR.var - Module global variables
```iecst
VAR
	bCtrl_ThR_CInc : BOOL; (*OldName: GAS_PLUS*)
	bCtrl_ThR_CDec : BOOL; (*OldName: GAS_MINUS*)
	bGnlWarning : BOOL; (*General warning*)
	bGnlTrip3 : BOOL; (*General trip*)
	bGnlTrip2 : BOOL; (*General trip*)
	bGnlTrip1 : BOOL; (*General trip*)
	bGnlTrip : BOOL; (*General trip*)
	Limit_Pinc : REAL; (* Limit value for load increase *)
	TimeSlot_Pinc : TIME; (* Time slot for monitoring any load increase *)
	xOpMode : OpMode; (*Used to determine the OpState of the engine*)
	bThR_Rel : BOOL; (* Thermal Reactor Release *)
	set_PT_KL_Pinc : BOOL := FALSE; (*set flap interval load increase*)
	FG_HEIZG_moduleTR : BOOL; (* Reaktor el. Heizung Ein *)
	bNoInitDetected : BOOL; (*always true, except 1cycle on init up*)
	IN_TR : IN_TR_Struct;
	MM2VIS : MM2VIS_Struct;
	VIS2MM : VIS2MM_Struct;
	OUT_TR : OUT_TR_Struct;
	ParaFactoryDefault : Para_Struct;
	Para : Para_Struct; (*Parameters*)
	pm : Para_Struct;
	pm1 : PERM_TR_Struct;
	TK_moduleTR : REAL; (* Temp. Reaktionskammer fuer Regelung *)
	TK1 : REAL; (* Temp. Reaktionskammer 1 *)
	TK2 : REAL; (* Temp. Reaktionskammer 2 *)
	xTRW06 : SR; (* Reaktor: Differenz TK1/TK2 max. *)
	xTRW05 : SR; (* Reaktor: Schaltschranktemp. max. *)
	xTRW04 : SR; (* Reaktor: Aufheizzeit ueberschr. *)
	xTRW08 : SR; (* Reaktor: Temp. Reakt.kammer min. *)
	xTRW07 : SR; (* Reaktor: Temp. Reakt.kammer max. *)
	bThR2_T_fault_ReactChamber : BOOL; (* Th.Reactor warning - reactor chamber temperature sensors failure - ThR2 *)
	xTRW02 : SR; (* Reaktor: Stoerung Druckluft *)
	xTRA02 : SR; (* Reaktor: Sicherheitsschleife *)
	xTRA01 : SR; (* Reaktor: Stoerg. Abgaskl. Mitte *)
	xTRW01 : SR; (* Reaktor: Fuehlerbruch *)
	xTRW03 : SR; (* Reaktor: Stoerg. Abgaskl. Ende *)
	xTON_INIT : TON;
	tCtrTR_Heater_In : _tGeACtrIn;
	tCtrTR_Heater_Out : _tGeACtrOut;
	xCtrTR_Heater : GeACtr; (*Controller instance*)
	RM_KL_END_AUS : BOOL;
	RM_KL_END_EIN : BOOL;
	KL_AUS_M_S : BOOL;
	KL_EIN_M_S : BOOL;
	xTRA01M : SR;
	bThR_RelTest : BOOL; (*!! Release thermoreactor for testing purpose only*)
	bThR_Failure : BOOL := 0; (* Thermoreactor failure *)
	bThR_elHeating : BOOL; (*Thermal reactor electrical heating ON*)
	bThr_AuxGasCompressor_Fault : BOOL;  (* Th.Reactor warning - auxiliary gas compressor fault *)
	bThr_AuxGasPr_PcheckFail : BOOL;  (* Th.Reactor warning - implausible auxiliary gas pressure before/after control valve *)
	bThR2_DPr_Hi : BOOL; (* Th.Reactor warning - differential pressure maximum - ThR2 *)
	bThR2_EH_gr1_T_blocked : BOOL; (* Th.Reactor electrical heating system - ThR2 - blocked status of heating element group 1 *)
	bThR2_EH_gr2_T_blocked : BOOL; (* Th.Reactor electrical heating system - ThR2 - blocked status of heating element group 2 *)
	bThR2_EH_gr3_T_blocked : BOOL; (* Th.Reactor electrical heating system - ThR2 - blocked status of heating element group 3 *)
	bThR2_EH_gr4_T_blocked : BOOL; (* Th.Reactor electrical heating system - ThR2 - blocked status of heating element group 4 *)
	bThR2_EH_gr5_T_blocked : BOOL; (* Th.Reactor electrical heating system - ThR2 - blocked status of heating element group 5 *)
	bThr2_AuxGasValve_fault : BOOL; (* Th.Reactor warning - auxiliary gas solenoid valve fault - ThR2 *)
	bThR2out_SCRin_DPr_Hi : BOOL; (* Exhaust aftertreatment warning - Thermal reactor outlet/SCR inlet high differential pressure - ThR2 *)
	bThr2_AuxGasValve_CtrlBlock : BOOL; (* Th.Reactor aux. gas heating system - ThR2 - aux. gas heating controller block due to valve closed *)
END_VAR
```

### Program Logical/ThermalReactor/GeneralTR (IEC) - General

#### GeneralTRCyclic.st - Cyclic code
```iecst
(*******************************************************************************
 GeneralTR	 			power limits and thresholds, controller increment/decrement, Operation hours, diagnostic visualization

This code is confidential AND proprietary to the INNIO Company.
It may NOT be used in any form, or reproduced in any manner,
without written permission of the INNIO Company.
Copyright, INNIO Company, 2019

Customized modifications: -
------------------------

History:
-------
V04.00.00.00	03-04-2014	Denk/Ganguly	new
V04.03.00.00	25-09-2014  Denk,			adjust step controller for Thermal reactor
				29-06-2015  Denk,			Operation hour for Reactor, Gas Injection and el. Heater
v04.09.00.00	20-02-2020 	Denk,			Thermalreactor failure added
V04.12.00.00	12-05-2022	Maran			bugfix: updated triggering signal for electrical heater operating hour counter
				12-07-2022	Maran			bugfix: included warning conditions TRW05, TRW06 and TRW07 for thermalreactor failure(W9309)
V04.13.00.00	28-11-2023	Maran			Added MM2VIS variables and warnings for thermal reactor auxiliary gas injection monitoring
V04.14.00.00	27-11-2024	Maran			Added Thermal reactor high differential pressure monitoring - ThR2,
											 included ThR2 temperature signal faults on left and right chamber for thermalreactor failure(W9309)
				27-11-2024	Maran			Added Thermal reactor auxiliary gas solenoid valve fault monitoring - ThR2,
											 added Thermal reactor outlet/SCR inlet high differential pressure monitoring

Instructions for use:
--------------------

Outstandings: -
------------

(*******************************************************************************)

PROGRAM _CYCLIC

	(* Operating mode *)
	xOpMode(in := IN_TR.iSt_OpMode);

	(* Check is power limit exceeded for Thermal Reactor *)
	xGR_MAXR_P_TRACT.In := IN_TR.rP_Act_Norm_Filt  * IN_TR.rP_Nom;
	xGR_MAXR_P_TRACT.Gw := Para.rP_Norm_ThR_Active * IN_TR.rP_Nom;    (* Default 48%  *)
	xGR_MAXR_P_TRACT.Hy := Para.rP_ThR_ActiveHy;                      (* Default 20kW *)
	xGR_MAXR_P_TRACT();

	(* Thermal Reactor release if Net parallel and power threshold crossed *)
	bThR_Rel := xOpMode.NetP AND IN_TR.tPB2MM.bParaSetupOk AND xGR_MAXR_P_TRACT.Q;

	(* ThermalReactor Main task: Thermocouple failure, pressurized air failure, valve end position failure, heat up failure, control panel high temperature,
								 high temperature difference within TK1 or TK2, reactor temperature maximum, minimum temperature, operating switch and emission monitoring active *)
	bThR_Failure := 	Para.bThR_Active
					AND bThR_Rel
					AND (xTRW01.Q1 OR bThR2_T_fault_ReactChamber OR xTRW02.Q1 OR xTRW03.Q1 OR xTRW04.Q1 OR xTRW05.Q1 OR xTRW06.Q1 OR xTRW07.Q1 OR xTRW08.Q1 OR NOT IN_TR.tThR_Swth_On.Di)
					AND	Para.iIdx_Em_AvgMon_Option > 0;

	(* Operation hour counter - Thermalreactor running *)
	xBH_OpHour_Reactor(enable := OUT_TR.bThR_Run, BH_adr := ADR(OpHour_Reactor.tick));
	xR_TRIG_OpHour_Reactor(CLK := xBH_OpHour_Reactor.BH_Imp);

	IF xR_TRIG_OpHour_Reactor.Q THEN	(* if an operation hour is finished *)
		(* operating hour counter *)
		VIS2MM.iCnt_OpHours_Reactor := VIS2MM.iCnt_OpHours_Reactor + 1;		(* increase counter *)
		(* check limits *)
		IF VIS2MM.iCnt_OpHours_Reactor >= 1000000000 THEN
			VIS2MM.iCnt_OpHours_Reactor := VIS2MM.iCnt_OpHours_Reactor - 1000000000;		(* check upper limit *)
		ELSIF VIS2MM.iCnt_OpHours_Reactor <= -1000000000 THEN
			VIS2MM.iCnt_OpHours_Reactor := VIS2MM.iCnt_OpHours_Reactor + 1000000000;		(* check lower limit *)
		END_IF;
	END_IF;

	(* Operation hour counter - Gas injection *)
	xBH_OpHour_GasInj(enable := OUT_TR.bThR_RelGas, BH_adr := ADR(OpHour_GasInj.tick));
	xR_TRIG_OpHour_GasInj(CLK := xBH_OpHour_GasInj.BH_Imp);

	IF xR_TRIG_OpHour_GasInj.Q THEN	(* if an operation hour is finished *)
		(* operating hour counter *)
		VIS2MM.iCnt_OpHours_GasInj := VIS2MM.iCnt_OpHours_GasInj + 1;		(* increase counter *)
		(* check limits *)
		IF VIS2MM.iCnt_OpHours_GasInj >= 1000000000 THEN
			VIS2MM.iCnt_OpHours_GasInj := VIS2MM.iCnt_OpHours_GasInj - 1000000000;		(* check upper limit *)
		ELSIF VIS2MM.iCnt_OpHours_GasInj <= -1000000000 THEN
			VIS2MM.iCnt_OpHours_GasInj := VIS2MM.iCnt_OpHours_GasInj + 1000000000;		(* check lower limit *)
		END_IF;
	END_IF;

	(* Operation hour counter - Electrical heater *)
	xBH_OpHour_Heater(enable := bThR_elHeating, BH_adr := ADR(OpHour_Heater.tick));
	xR_TRIG_OpHour_Heater(CLK := xBH_OpHour_Heater.BH_Imp);

	IF xR_TRIG_OpHour_Heater.Q THEN	(* if an operation hour is finished *)
		(* operating hour counter *)
		VIS2MM.iCnt_OpHours_Heater := VIS2MM.iCnt_OpHours_Heater + 1;		(* increase counter *)
		(* check limits *)
		IF VIS2MM.iCnt_OpHours_Heater >= 1000000000 THEN
			VIS2MM.iCnt_OpHours_Heater := VIS2MM.iCnt_OpHours_Heater - 1000000000;		(* check upper limit *)
		ELSIF VIS2MM.iCnt_OpHours_Heater <= -1000000000 THEN
			VIS2MM.iCnt_OpHours_Heater := VIS2MM.iCnt_OpHours_Heater + 1000000000;		(* check lower limit *)
		END_IF;
	END_IF;

	(*  Thermal reactor auxiliary gas injection monitoring *)
	IF Para.bThR_auxGasMonitor THEN
		(* definition of running status for Th.Reactor aux.gas compressor *)
		MM2VIS.bThr_AuxGasCompressor_Run := OUT_TR.bThR_RelGas AND ((IN_TR.tPr_ThR_AuxGasBeforeCV.Ai >= rPr_ThR_AuxGas_thres_ComprRun) OR
		(MM2VIS.bThr_AuxGasCompressor_Run AND (IN_TR.tPr_ThR_AuxGasBeforeCV.Ai >= rPr_ThR_AuxGas_thres_ComprRun - rPr_ThR_AuxGas_thres_ComprRunHy)));

		(* calculation of Th.Reactor aux.gas differential pressure *)
		MM2VIS.rPr_Diff_ThR_AuxGasCV := IN_TR.tPr_ThR_AuxGasBeforeCV.Ai - IN_TR.tPr_ThR_AuxGasAfterCV.Ai;

		(* calculation of estimated Th.Reactor aux.gas volume flow *)
		IF MM2VIS.bThr_AuxGasCompressor_Run THEN
			MM2VIS.rFlow_ThR_AuxGasCV := (MAX(0, IN_TR.tPos_ThR_AuxGasCV_Act.Ai) * (514 * Para.rThR_auxGasCV_Kv)) / SQRT((1.24 * 338.15) / LIMIT( 0.00001, (MAX(0, (MM2VIS.rPr_Diff_ThR_AuxGasCV / 1000)) * ((IN_TR.tPr_ThR_AuxGasAfterCV.Ai / 1000) + 1.01325)), 10)) ;
		ELSE
			MM2VIS.rFlow_ThR_AuxGasCV := 0;
		END_IF
	ELSE
		MM2VIS.bThr_AuxGasCompressor_Run := FALSE;
		MM2VIS.rPr_Diff_ThR_AuxGasCV := 0;
		MM2VIS.rFlow_ThR_AuxGasCV := 0;
	END_IF
	(* Th.Reactor warning - auxiliary gas compressor fault *)
	xTON_ThR_AuxGasCompr_Fault(IN := Para.bThR_auxGasMonitor AND OUT_TR.bThR_RelGas AND NOT MM2VIS.bThr_AuxGasCompressor_Run AND IN_TR.tPr_ThR_AuxGasBeforeCV.GoodQual, PT := tiTON_ThR_AuxGasCompr_Fault);
	bThr_AuxGasCompressor_Fault := xTON_ThR_AuxGasCompr_Fault.Q;
	(* Th.Reactor warning - implausible auxiliary gas pressure before/after control valve *)
	xTON_ThR_AuxGasPr_PcheckFail(IN := Para.bThR_auxGasMonitor AND OUT_TR.bThR_RelGas AND (IN_TR.tPr_ThR_AuxGasAfterCV.Ai >= rPr_ThR_AuxGas_thres_ComprRun) AND (MM2VIS.rPr_Diff_ThR_AuxGasCV < 0) AND
	 IN_TR.tPr_ThR_AuxGasBeforeCV.GoodQual AND IN_TR.tPr_ThR_AuxGasAfterCV.GoodQual AND (NOT Para.bThR2_Ena OR OUT_TR.tThR2_AuxGasShutOffValve_Dem.Do), PT := tiTON_ThR_AuxGasPr_PcheckFail);
	bThr_AuxGasPr_PcheckFail := xTON_ThR_AuxGasPr_PcheckFail.Q;

	(* Thermal reactor high differential pressure monitoring - ThR2 *)
	MM2VIS.rPr_Diff_ThR2 := IN_TR.tPr_ThR2_Inlet.Ai - IN_TR.tPr_ThR2_Outlet.Ai;
	xTON_ThR2_DPr_Hi(IN := Para.bThR2_Ena AND IN_TR.tPr_ThR2_Inlet.GoodQual AND IN_TR.tPr_ThR2_Outlet.GoodQual AND (MM2VIS.rPr_Diff_ThR2 > rDPr_ThR2_thres_Hi), PT := tiTON_ThR2_DPr_Hi);
	bThR2_DPr_Hi := xTON_ThR2_DPr_Hi.Q;

	(* Thermal Reactor auxiliary gas solenoid valve fault monitoring - ThR2 *)
	IF EDGENEG(OUT_TR.tThR2_AuxGasShutOffValve_Dem.Do) THEN // record aux.gas pressure value at solenoid valve closing
		IF ((MM2VIS.rPr_Diff_ThR_AuxGasCV  >= rPr_ThR2_AuxGasValve_mon_inc + rPr_ThR2_AuxGasValve_mon_delta) AND IN_TR.tPr_ThR_AuxGasBeforeCV.GoodQual AND IN_TR.tPr_ThR_AuxGasAfterCV.GoodQual) THEN
			rPr_ThR2_AuxGasValve_mon_ref := IN_TR.tPr_ThR_AuxGasAfterCV.Ai;
			rPr_ThR2_AuxGasValve_mon_BefCV := IN_TR.tPr_ThR_AuxGasBeforeCV.Ai;
			bThR2_AuxGasValve_mon_valid := TRUE;
		ELSE
			bThR2_AuxGasValve_mon_valid := FALSE;
		END_IF
	END_IF
	xTOF_Thr2_AuxGasValve_mon_valid(IN := EDGENEG(OUT_TR.tThR2_AuxGasShutOffValve_Dem.Do), PT := tiTON_Thr2_AuxGasValve_fault + T#500ms);
	IF (NOT OUT_TR.bThR_RelGas) OR (NOT xTOF_Thr2_AuxGasValve_mon_valid.Q) THEN //reset aux. gas solenoid valve fault monitoring if aux. gas system is stopped or check valid timer is elapsed
		bThR2_AuxGasValve_mon_valid := FALSE;
	END_IF
	xTON_Thr2_AuxGasValve_fault(IN := bThR2_AuxGasValve_mon_valid AND MM2VIS.bThr_AuxGasCompressor_Run AND NOT OUT_TR.tThR2_AuxGasShutOffValve_Dem.Do AND			(*pressure verification made during close command for aux. gas solenoid valve*)
	 ((IN_TR.tPr_ThR_AuxGasAfterCV.Ai <= rPr_ThR2_AuxGasValve_mon_ref + rPr_ThR2_AuxGasValve_mon_inc) AND IN_TR.tPr_ThR_AuxGasAfterCV.GoodQual) AND					(*pressure after CV - pressure increase verification*)
	 ((IN_TR.tPr_ThR_AuxGasBeforeCV.Ai >= rPr_ThR2_AuxGasValve_mon_BefCV - 0.6 * rPr_ThR2_AuxGasValve_mon_delta) AND IN_TR.tPr_ThR_AuxGasBeforeCV.GoodQual) AND		(*pressure before CV not decreased during the verification*)
	 ((IN_TR.tPos_ThR_AuxGasCV_Act.Ai >= rPos_ThR2_AuxGasValve_mon_valid) AND IN_TR.tPos_ThR_AuxGasCV_Act.GoodQual), PT := tiTON_Thr2_AuxGasValve_fault);			(*CV open position during the pressure verification*)
	bThr2_AuxGasValve_fault := xTON_Thr2_AuxGasValve_fault.Q;

	(* Exhaust aftertreatment: Thermal reactor outlet/SCR inlet high differential pressure monitoring - ThR2*)
	IF Para.bThR2_Ena AND ((Para.bSCR_Active OR Para.bSCR_Cust_Active) AND Para.bPr_SCR_CatIn_Exist) THEN
		MM2VIS.rPr_Diff_ThR2out_SCRin := IN_TR.tPr_ThR2_Outlet.Ai - (IN_TR.tPr_SCR_CatIn.Ai * 1000);
	ELSE
		MM2VIS.rPr_Diff_ThR2out_SCRin := 0;
	END_IF
	xTON_ThR2out_SCRin_DPr_Hi(IN := (MM2VIS.rPr_Diff_ThR2out_SCRin >= rDPr_ThR2_SCR_thres_Hi) AND IN_TR.tPr_ThR2_Outlet.GoodQual AND IN_TR.tPr_SCR_CatIn.GoodQual, PT := tiTON_ThR2out_SCRin_DPr_Hi);
	bThR2out_SCRin_DPr_Hi := xTON_ThR2out_SCRin_DPr_Hi.Q;

END_PROGRAM
```

#### GeneralTR.var - Local variables
```iecst
VAR
	xGR_MAXR_P_TRACT : GR_MAXR;
	xBH_OpHour_GasInj : BH;
	xR_TRIG_OpHour_GasInj : R_TRIG;
	OpHour_GasInj : bh_typ;
	xBH_OpHour_Reactor : BH;
	xR_TRIG_OpHour_Reactor : R_TRIG;
	OpHour_Reactor : bh_typ;
	xBH_OpHour_Heater : BH;
	xR_TRIG_OpHour_Heater : R_TRIG;
	OpHour_Heater : bh_typ;
	rPr_ThR_AuxGas_thres_ComprRun : REAL := 140; (* Thermal reactor - auxiliary gas pressure threshold for compressor running status display [mbar] *)
	rPr_ThR_AuxGas_thres_ComprRunHy : REAL := 10; (* Thermal reactor - hysteresis for auxiliary gas pressure for compressor running status [mbar] *)
	xTON_ThR_AuxGasCompr_Fault : TON; (* TON delay for Th.Reactor warning - auxiliary gas compressor fault *)
	tiTON_ThR_AuxGasCompr_Fault : TIME := T#20s; (* Auxiliary timer variable *)
	xTON_ThR_AuxGasPr_PcheckFail : TON; (* TON delay for Th.Reactor warning - implausible auxiliary gas pressure before/after control valve *)
	tiTON_ThR_AuxGasPr_PcheckFail : TIME := T#10s; (* Auxiliary timer variable *)
	rDPr_ThR2_thres_Hi : REAL := 25.0; (* Thermal reactor maximum differential pressure threshold [mbar] *)
	xTON_ThR2_DPr_Hi : TON; (* TON delay for Th.Reactor warning - differential pressure maximum - ThR2 *)
	tiTON_ThR2_DPr_Hi : TIME := T#10s; (* Auxiliary timer variable *)
	rPr_ThR2_AuxGasValve_mon_ref : REAL; (* Thermal reactor - auxiliary gas solenoid valve monitoring - pressure verification reference [mbar] *)
	rPr_ThR2_AuxGasValve_mon_BefCV : REAL; (* Thermal reactor - auxiliary gas solenoid valve monitoring - pressure reference before control valve [mbar] *)
	rPr_ThR2_AuxGasValve_mon_inc : REAL := 30; (* Thermal reactor - auxiliary gas solenoid valve monitoring - expected pressure increase after CV at valve closing [mbar] *)
	rPr_ThR2_AuxGasValve_mon_delta : REAL := 10; (* Thermal reactor - auxiliary gas solenoid valve monitoring - tolerance value for pressure verification [mbar] *)
	bThR2_AuxGasValve_mon_valid : BOOL; (* Thermal reactor - auxiliary gas solenoid valve monitoring valid *)
	rPos_ThR2_AuxGasValve_mon_valid : REAL := 0.20; (* Thermal reactor - auxiliary gas solenoid valve monitoring - minimum CV position for pressure verification validity [%] *)
	xTON_Thr2_AuxGasValve_fault : TON; (* TON delay for Th.Reactor warning - auxiliary gas solenoid valve fault *)
	xTOF_Thr2_AuxGasValve_mon_valid : TOF; (* TOF timer for Th.Reactor - auxiliary gas solenoid valve monitoring valid *)
	tiTON_Thr2_AuxGasValve_fault : TIME := T#3s; (* Auxiliary timer variable *)
	rDPr_ThR2_SCR_thres_Hi : REAL := 30.0; (* Exhaust aftertreatment - Thermal reactor outlet/SCR inlet maximum differential pressure threshold [mbar] *)
	xTON_ThR2out_SCRin_DPr_Hi : TON; (* TON delay for Exhaust aftertreatment warning - Thermal reactor outlet/SCR inlet high differential pressure *)
	tiTON_ThR2out_SCRin_DPr_Hi : TIME := T#10s; (* Auxiliary timer variable *)
END_VAR
```

### Program Logical/ThermalReactor/reac_set (IEC) - Settings

#### reac_setCyclic.st - Cyclic code
```iecst
(*******************************************************************************
reac_set	THERMOREACTOR SETTINGS

This code is confidential AND proprietary TO the INNIO Company.
It may NOT be used in any form, or reproduced in any manner,
without the express written permission OF the INNIO Company.
Copyright, INNIO Company, 2019

Customized modifications: -
------------------------

History:
-------
V3.20.0 16-12-2010  Thaler, generated
        16-12-2010	Thaler, last modification,
                            compatible with XT Version from V2.2x upwards.

V04.00.00	04-04-2014  Ganguly, converted to modular software

Instructions for use:
--------------------
description interface --> Task "reactor" ( BOOL, where NOT otherwise stated ):

(* UM_E_NEU_moduleTR:       type of position switches 4-way-flap: TRUE = 3 end positions (5 switches)
sel_NatGas:     select gas injection natural gas (spare)
sel_woGas:      select w/o gas injection
TK_w_woGas:     TK_moduleTR setpoint without gas injection  ( 0,1 °C   )
PT_KL_Pinc:     flap switching interval load incr. ( 1,0 sec. )
set_PT_KL_Pinc: set flap interval load increase

Outstandings: -
------------
*******************************************************************************)

PROGRAM _CYCLIC

IF Para.bThR_woGas THEN
    (* thermal reactor - TK_moduleTR setpoint without gas injection *)
  	(* --> check/choose Reserve Parameter No. plant specific ! *)
    (* Old Parameter: TK_w_woGas. Default 720.0°C *)
    Para.rT_ThR_SetwoGas := LIMIT (700.0, Para.rT_ThR_SetwoGas, 780.0); (* 0,1°C *)

    (* thermal reactor - limit value for load increase within the time slot *)
	(* --> check/choose Reserve Parameter No. plant specific ! *)
	Limit_Pinc := LIMIT (20.0, Para.rT_ThR_LimPInc, 80.0); (* 0,1 % *)

    (* thermal reactor - time slot for monitoring any load increase *)
	(* --> check/choose Reserve Parameter No. plant specific ! *)
    TimeSlot_Pinc := LIMIT (T#600s, Para.ti_ThR_TimePInc, T#1000s); (* 1,0 sec *)

	No_ScanIntervals := LIMIT (6, (TIME_TO_INT(TimeSlot_Pinc)/ 10), 100);

    (* thermal reactor - duration for set the flap switching interval on load increase value *)
	(* --> check/choose Reserve Parameter No. plant specific ! *)
	// Old Parameter PTOF_KL_Pinc_i. Para.ti_ThR_ValDurationPInc = T#600s (default)
    Para.ti_ThR_ValDurationPInc := LIMIT (T#60s, Para.ti_ThR_ValDurationPInc, T#3600s); (* 1,0 sec *)

    (* thermal reactor - flap switching interval: load increase value *)
	(* --> check/choose Reserve Parameter No. plant specific ! *)
    // Old Parameter PT_KL_Pinc. Para.ti_ThR_ValIntervalPInc = T#210s (default)
    Para.ti_ThR_ValIntervalPInc := LIMIT (T#100s, Para.ti_ThR_ValIntervalPInc, T#600s); (* 1,0 sec *)

END_IF;

(* Takt 1 sec. *)
xTOF_TAKT02(IN:= xTON_TAKT01.Q, PT:= T#350ms);
xTON_TAKT01(IN:= NOT xTOF_TAKT02.Q, PT:= T#350ms);
xR_TRIG_TAKT1(CLK:= xTON_TAKT01.Q);
TAKT1 := xR_TRIG_TAKT1.Q;
(* Takt 10 sec. *)
xTOF_TAKT102(IN:= xTON_TAKT101.Q, PT:= T#9s350ms);
xTON_TAKT101(IN:= NOT xTOF_TAKT102.Q, PT:= T#350ms);
xR_TRIG_TAKT10(CLK:= xTON_TAKT101.Q);
TAKT10 := xR_TRIG_TAKT10.Q;

(* Ringbuffer *)
IF TAKT10 = TRUE THEN (* scan interval *)
    Delta_P := IN_TR.rP_Act_Norm_Filt - P_old; (* load delta within scan interval, 0,1 % *)
    P_old   := IN_TR.rP_Act_Norm_Filt;
    IF (FG_HEIZG_moduleTR = TRUE OR IN_TR.tGCB_On.Di) THEN
        DeltaP[i1] := Delta_P; (* 0,1 % *)
    ELSE
        DeltaP[i1] := 0; (* 0,1 % *)
    END_IF;
    i1 := i1 +1;
    IF i1 > (No_ScanIntervals - 1) THEN
        i1 := 0;
    END_IF;
END_IF;

a := 0;
FOR i := 0 TO (No_ScanIntervals - 1) BY 1 DO
    a := a + DeltaP[i];
END_FOR;
DeltaP_t := a; (* load delta within time slot, 0,1 % *)

(* set the flap switching interval on load increase value. Old signal PTOF_KL_Pinc*)
xTOF_KL_Pinc(IN:= (DeltaP_t >= Limit_Pinc), PT:= Para.ti_ThR_ValDurationPInc);

(* interface --> Task "reactor" *)
set_PT_KL_Pinc := xTOF_KL_Pinc.Q;

(* end of settings *)
(******************************************************************************)
END_PROGRAM
```

#### reac_setInit.st - Initialization code
```iecst
(********************************************************************
 * COPYRIGHT -- INNIO Company
 ********************************************************************
 * Program: reac_set
 * File: reac_setInit.st
 * Author: thalerjo
 * Created: November 18, 2010
 ********************************************************************
 * Implementation of program reac_set
 ********************************************************************)

PROGRAM _INIT

(* TODO : Add your code here *)

END_PROGRAM
```

#### reac_set.var - Local variables
```iecst
(********************************************************************
 * COPYRIGHT -- INNIO Company
 ********************************************************************
 * Program: reac_set
 * File: reac_set.var
 * Author: thalerjo
 * Created: November 18, 2010
 ********************************************************************
 * Local variables of program reac_set
 ********************************************************************)
VAR
	TAKT10 : BOOL;
	TAKT1 : BOOL;
	No_ScanIntervals : INT;
	i1 : INT;
	i : INT;
	P_old : REAL;
	a : REAL;
	Delta_P : REAL;
	DeltaP_t : REAL;
	DeltaP : ARRAY[0..99] OF REAL;
	xR_TRIG_TAKT10 : R_TRIG;
	xR_TRIG_TAKT1 : R_TRIG;
	xTOF_TAKT102 : TOF;
	xTOF_TAKT02 : TOF;
	xTOF_KL_Pinc : TOF;
	xTON_TAKT101 : TON;
	xTON_TAKT01 : TON;
END_VAR
```

### Program Logical/ThermalReactor/reactor (IEC) - Main task
